(* CoDeSys 2.3.9.31 project: BA17xx.pro *)
(* Libraries: TcBaseMath.lib 27.7.04 13:07:56, TcMC2_Camming.lib 11.12.14 09:45:00, TcMath.lib 23.9.04 16:15:30, TcNC.lib 10.10.08 18:55:34, TcBase.lib 14.5.09 13:14:08, TcMC2.lib 22.12.11 16:37:48, TcSystem.lib 9.3.10 11:21:30, TcXmlDataSrv.lib 29.9.06 15:13:00, TcUtilities.lib 7.4.10 10:22:08, COMlibV2.lib 1.8.08 14:22:48, TcRFID.lib 20.9.10 12:18:58, STANDARD.LIB 5.6.98 13:03:02, TcCX1000System.lib 11.10.10 12:52:26, TcEtherCAT.lib 15.1.10 20:43:56, TcTestAndSet.lib 23.2.09 13:50:08, TcDrive.lib 17.3.10 13:50:30, TcMc2Drive.lib 19.1.10 11:34:38, TcIoFunctions.lib 21.7.11 17:19:20 *)

(* Global variable list: EPT Lib/Global_Checks *)
VAR_GLOBAL
	CheckBounds_ErrCnt 			: DINT := 0;
	CheckByteZeroDiv_ErrCnt 		: DINT := 0;
	CheckDWordZeroDiv_ErrCnt 	: DINT := 0;
	CheckRealZeroDiv_ErrCnt 		: DINT := 0;
	CheckWordZeroDiv_ErrCnt 		: DINT := 0;
	CheckRangeSigned_ErrCnt		: DINT := 0;
	CheckRangeUnsigned_ErrCnt	: DINT := 0;
END_VAR

(* Global variable list: Global_Visu *)
VAR_GLOBAL
	visu 			: 	struct_visu;
	visu_hinten	:	struct_visu_hinten;
END_VAR

(* Global variable list: Globale_Achsen *)
VAR_GLOBAL
	(* Achsen *)
	z_achse								: AXIS_REF;
	axis_z_achse							: struct_achse;

	bestueckachse						: AXIS_REF;
	axis_bestueckachse					: struct_achse;

	virtuelle_master_achse					: AXIS_REF;
	axis_virt_master						: struct_achse;

	getriebe_einstell_achse					: AXIS_REF;

	y_achse								: AXIS_REF;
	axis_y_achse							: struct_achse;

	b_achse								: AXIS_REF;
	axis_bandeinzug_achse				: struct_achse;

	transport_wt_achse					:AXIS_REF;
	axis_transport_wt_achse				: struct_achse;
END_VAR

(* Global variable list: Globale_IO *)
VAR_GLOBAL
	(* =====SMEMA -Schnittstelle===== *)
	(* Digitale IO *)
	(* SMEMA -Schnittstelle *)
	e_smema_station_vorher_in_anforderung			AT %I* : BOOL;
	e_smema_station_vorher_in_abgegeben			AT %I* : BOOL;
	a_smema_station_vorher_out_erlaubnis			AT %Q* : BOOL;
	a_smema_station_vorher_out_angekommen		AT %Q* : BOOL;

	e_smema_station_nachher_in_erlaubnis			AT %I* : BOOL;
	e_smema_station_nachher_in_angekommen		AT %I* : BOOL;
	a_smema_station_nachher_out_anforderung		AT %Q* : BOOL;
	a_smema_station_nachher_out_abgegeben		AT %Q* : BOOL;

	(* ADS-Kommunikation *)
	st_ads_smema_station_vorher					: struct_station_vorher;
	st_ads_smema_station_nachher					: struct_station_nachher;

	(* Bandwechselvorschub/Rasterfolienvorschub *)
	a_zyl_vorschub_einfahren						AT %Q* : BOOL;
	a_zyl_vorschub_ausfahren						AT %Q* : BOOL;

	(* Fänger Rasterfolie/Bandeinzug bzw. Klemmen Rasterfolie/Bandeinzug *)
	a_zyl_faenger_einfahren						AT %Q* : BOOL;
	a_zyl_klemmen_einfahren						AT %Q* : BOOL;
END_VAR

(* Global variable list: EPT Lib/Globale_Var *)
VAR_GLOBAL
	gi16_betriebsart					: enum_betriebsarten;
END_VAR

VAR_GLOBAL PERSISTENT
	gst_system_time					: TIMESTRUCT;
	gdt_system_time					: DT;
	gstr_system_time				: STRING;
	b_system_time_valid				: BOOL;
	gstr_datum						: STRING;
	gstr_uhrzeit						: STRING;
END_VAR

VAR_GLOBAL CONSTANT
	MAX_NOCKENGERUEST			: INT := 63;
END_VAR

(* Global variable list: Globale_Var_BA *)
VAR_GLOBAL
	garr_stoermeldungen				: ARRAY[0..4999] OF BOOL;
	garr_betriebsmeldungen			: ARRAY[0..4999] OF BOOL;

	gb_ba_auto_kontroller				: BOOL;
	gi16_maschinenstatusinfo			: enum_maschinenstatus;
	gb_nach_bawe_einzelfertigung		: BOOL := FALSE;
	gi16_anzahl_Teile_autostop_bandwechsel	: INT := 0;

	bbgen							: struct_objekt;
	wartung							: struct_objekt;
	bandspruehoeler					: struct_objekt;
	haspel_re						: struct_haspel_V2;
	haspel_li							: struct_haspel_V2;
	betriebsarten						: struct_betriebsarten;
	bandeinzug_kontroller				: struct_objekt;
	bandwechsel_kontroller			: struct_bandwechsler;
	haspel_kontroller					: struct_haspelkontroller;
	stoerungen_quittieren				: struct_objekt;
	betriebsfreigaben					: struct_betriebsfreigaben;
	betriebsstundenzaehler			: struct_betriebsstundenzaehler;
	wkz_absicherung					: struct_objekt;
	stueckzahlen						: struct_stueckzahl;
	balluff_tag_reader					: struct_balluff_tag_reader;
	barcode							: struct_barcode;
	hublift_links						: struct_objekt;
	hublift_rechts						: struct_objekt;
	wt_transport_kontroller				: struct_objekt;
	wt_transport_beladen				: struct_objekt;
	wt_transport_warteposition_1700		: struct_objekt;
	wt_transport_beladen_achse_1700	: struct_objekt;
	wt_transport_beladen_1720			: struct_objekt;
	wt_transport_warteposition_1720		: struct_objekt;
	wt_transport_abgabe				: struct_objekt;
	safety							: struct_objekt;
	xml_server						: struct_objekt;
	fb_edit_mfps_bestuecken_z			: struct_mf_editor;
	fb_edit_mfps_bestuecken_y			: struct_mf_editor;
	fb_edit_mfps_bestuecken_b		: struct_mf_editor;
	fb_edit_mfps_yz_tisch	 			: struct_mf_editor;
	fb_edit_mfps_bestueckachse		: struct_mf_editor;
	fb_camtable_bestueckachse		: struct_camtable_maker;
	(*rasterplattenmontage				: struct_objekt;
	rasterplattenwendestation			: struct_objekt;
	ruettler_rasterplatte				: struct_rapl_ruettler;*)
	einpresskraft_kontroller				: struct_objekt;
	kraftmessdose					: struct_analogin;
	nockenschaltwerk_bestueckachse	: struct_nockenschaltwerk_lreal;
	routing_backpanel					: struct_objekt;
	routing_nachbarpc					: struct_objekt;
	ads_kommu_pc_vorher			: struct_ads_kommunikation;
	ads_kommu_pc_nachher			: struct_ads_kommunikation;
	rasterfolienmontage				: struct_objekt;
	rasterfolieneinzug					: struct_objekt;
	edit_mfps						: struct_objekt;
	Lesen_Schreiben_Tag				: struct_objekt;
	Service							: struct_objekt;

	UPS							: struct_objekt;

	st_ctrl_in_empty					:struct_ctrl_in;
	st_ctrl_out_empty				:struct_ctrl_out;

	(* Daten welche vom Tag gelesen / zum Tag geschrieben werden *)
	gst_tag_data						: struct_tag_data;

	gi16_bbgen_auftrag				: enum_bbgen_auftrag := KEIN_BB_AUFTRAG;
	gi16_wartung_auftrag				: enum_wartung_auftrag :=  KEIN_WARTUNG_AUFTRAG;

	gst_bestueckbild					: struct_bestueckbild;
	gst_bestueckbild_halbauto			: struct_bestueckbild_halbauto;
	s_alte_artikelnummer				: STRING(50) := '';

	(* Version *)
	gs_version						: STRING := '*.zip';
	lr_debug : LREAL;

	(* Datenstruktur der Werkzeuge und STV auf der Maschine, welche per XML-File auf der Festplatte abgespeichert werden *)
	gst_datensatz						: struct_datensatz;

	(* Barcodedaten *)
	gst_barcode_daten				: struct_barcode_daten;

	gb_memEndOfBandMarkNIO		: BOOL := FALSE;	(*
	Diese Änderung wurde 1:1 aus Tschechien übernommen.
	Merker "gb_memEndOfBandMarkNIO" für Bandende während des Bestückens. Diese Variable gilt nur
	für den One27 in Tschechien. Während des Bestückens wird der Bandende Sensor abgefragt. Wenn
	noch mehr wie 80 Pins zu bestücken sind und der Bandende Sensor anschlägt, wird ein "HALT_AXIS"
	der virtuellen Masterachse ausgeführt. Die Achse bleibt zufällig irgendwo stehen. Der WT bleibt auf
	Bestückposition stehen. Eine Fehlermeldung kommt vom Bandwechselkontroller. Dann muss die 
	Anlage quittiert werden. Bestückachse fährt in Grundstellung und WT fährt auf Übergabeposition.
	Danach wird der Bandwechselvorgang gestartet. *)

	EtherCatDiag						:ARRAY[1..MaxNoOfMaster] OF FB_EtherCatDiag;
END_VAR

VAR_GLOBAL PERSISTENT
	(* manuelles Bestückbild *)
	gst_manuelles_bestueckprogramm	: struct_bestueckprogramm;
	gst_PersDaten						: struct_PD;
END_VAR
VAR_GLOBAL CONSTANT
	MaxNoOfMaster					:INT:=4;(*Maximale Anzahl Master für Ethercat Diagnose*)
	MaxNoOfSlaves					:INT:=40;(*Maximale Anzahl Slaves für Ethercat Diagnose*)
	MaxNoOfWkz						:INT:=24;(*Maximale Anzahl an Werkzeuge*)
END_VAR

(* Global variable list: Globale_XML_Server *)
VAR_GLOBAL
	(* Initialisierung der zu schreibenden Variablen in dem XML-File *)
	gs_xml_laufwerk					: STRING := 'D:\';
	gs_xml_path_root				: STRING := 'BBGen';
	gs_xml_path_md					: STRING(255) := 'MD';
	gs_xml_dateiname_md			: STRING := 'Maschinendaten';
	gs_xml_path_wkz				: STRING := 'WKZ';
	gs_xml_datei_erweiterung		: STRING := '.xml';
	gs_xml_symname_wkz			: STRING := 'gst_datensatz.st_wkz';
	gs_xml_symname_md			: STRING := 'gst_datensatz.st_md';
	s_PLC_name					: STRING(255);
	s_PLC_path						: STRING(255);
	s_Projekt_path					: STRING(255);

	(* Pfadnamen für Daten (ohne Laufwerksangabez.B."C:\_Datensatz" wird der Projektpfad angehängt)*)
	s_tools_path					: STRING(255):='Tools\';
	s_md_path 						: STRING(255):='MD\';

END_VAR

(* Global variable list: Globale_Zylinder *)
VAR_GLOBAL
	(* Gemeinsam *)
	zyl_wt_zentrierer_tisch				: struct_st_zylinder;
	zyl_wt_stopper_tisch				: struct_st_zylinder;
	zyl_wt_stopper_auslauf				: struct_st_zylinder;

	zyl_haspel_re_heben				: struct_st_zylinder;
	zyl_haspel_re_abspulen			: struct_st_zylinder;
	zyl_haspel_li_heben				: struct_st_zylinder;
	zyl_haspel_li_abspulen			: struct_st_zylinder;
	zyl_haspel_re_sperren				: struct_st_zylinder;
	zyl_haspel_li_sperren			:	 struct_st_zylinder;

	zyl_hublift_rechts_lift				: struct_st_zylinder;
	zyl_hublift_rechts_wt_einzug			: struct_st_zylinder;
	zyl_hublift_rechts_wt_klinke			: struct_st_zylinder;
	zyl_hublift_links_lift					: struct_st_zylinder;
	zyl_hublift_links_wt_einzug			: struct_st_zylinder;
	zyl_hublift_links_wt_klinke			: struct_st_zylinder;
	zyl_hublift_links_stopper			: struct_st_zylinder;
	zyl_hublift_links_eingriffschutz		: struct_st_zylinder;

	(* BSH 1700 *)
	zyl_bandfaenger					: struct_st_zylinder;
	zyl_bandklemmen					: struct_st_zylinder;
	zyl_bawe_vorschub				: struct_st_zylinder;
	zyl_bawe_querschub				: struct_st_zylinder;
	zyl_bawe_faenger_li				: struct_st_zylinder;
	zyl_bawe_faenger_re				: struct_st_zylinder;
	zyl_bawe_halter_li					: struct_st_zylinder;
	zyl_bawe_halter_re				: struct_st_zylinder;
	zyl_haspel_verschieben			: struct_st_zylinder;
	zyl_bandeinzuege_verschieben		: struct_st_zylinder;
	zyl_oelen_unten				: struct_st_zylinder;
	zyl_oelen_oben				: struct_st_zylinder;
	zyl_Indexier_Bestueckpos			: struct_st_zylinder;
	zyl_Indexier_Einlauf				: struct_st_zylinder;

	(* Rasterplatte *)
(*	zyl_rapl_aufpressen				: struct_st_zylinder;
	zyl_rapl_schacht					: struct_st_zylinder;
	zyl_rapl_kontaktfuehrung			: struct_st_zylinder;
	zyl_rap_ausschieben				: struct_st_zylinder;
	zyl_rapl_einschieben				: struct_st_zylinder;*)

	(* BSV1720 *)
	zyl_wt_stopper_einlauf				: struct_st_zylinder;
	zyl_bandfaenger_li				: struct_st_zylinder;
	zyl_bandfaenger_re				: struct_st_zylinder;
	zyl_bandklemmen_li				: struct_st_zylinder;
	zyl_bandklemmen_re				: struct_st_zylinder;

	(* Rasterfolie *)
	zyl_rafo_faenger					: struct_st_zylinder;
	zyl_rafo_klemmen					: struct_st_zylinder;
	zyl_rafo_vorschub					: struct_st_zylinder;
	zyl_rafo_kamm					: struct_st_zylinder;
	zyl_rafo_vorzentrierer				: struct_st_zylinder;
END_VAR

(* Global variable list: TwinCAT_Configuration *)
(* Generated automatically by TwinCAT - (read only) *)
VAR_CONFIG
	ST_AbfallBlasluft.a_AbfallBlasluft AT %QX5.0 : BOOL;
	ST_Bandeinzug_Kontroller_1700.e_wc_state AT %IX1272.0 : BOOL;
	ST_Bandeinzug_Kontroller_1700.e_gls_bandvorschubkontrolle AT %IX16.0 : BOOL;	(*  ~ {LinkedWith:TIID^Gerät 1 (EtherCAT)^A160 (EP2338-0001)^Channel 3^ST_Rasterfolienmontage.e_rasterfolie_aufgepresst} *)
	ST_Bandeinzug_Kontroller_1720.e_ls_bandende_re AT %IX16.1 : BOOL;
	ST_Bandeinzug_Kontroller_1720.e_ls_bandende_li AT %IX16.2 : BOOL;
	ST_Bandeinzug_Kontroller_1720.e_wc_state AT %IX1272.1 : BOOL;
	ST_Bandeinzug_Kontroller_1720.e_gls_bandvorschubkontrolle_li AT %IX820.0 : BOOL;
	ST_Bandeinzug_Kontroller_1720.e_gls_bandvorschubkontrolle_re AT %IX820.1 : BOOL;
	ST_BandoelerZylinder.a_ventil_oben AT %QX1144.0 : BOOL;	(*  ~ {LinkedWith:TIID^Gerät 1 (EtherCAT)^A170 (EP2338-0001)^Channel 15^ST_BandoelerZylinder.a_ventil_oben} *)
	ST_BandoelerZylinder.a_ventil_unten AT %QX1144.1 : BOOL;	(*  ~ {LinkedWith:TIID^Gerät 1 (EtherCAT)^A170 (EP2338-0001)^Channel 16^ST_BandoelerZylinder.a_ventil_unten} *)
	ST_BandoelerZylinder.e_fuellstand AT %IX1280.0 : BOOL;	(*  ~ {LinkedWith:TIID^Gerät 1 (EtherCAT)^A38 Transportsystem (EP2338-0001)^Channel 8^ST_Menzel_Spruehoeler.e_fuellstand} *)
	ST_BandoelerZylinder.e_druck_oelbehaelter AT %IX1280.1 : BOOL;	(*  ~ {LinkedWith:TIID^Gerät 1 (EtherCAT)^A38 Transportsystem (EP2338-0001)^Channel 7^ST_Menzel_Spruehoeler.e_druck_oelbehaelter} *)
	ST_Bandwechsel_Kontroller.e_ls_bandende_li AT %IX16.4 : BOOL;	(*  ~ {LinkedWith:TIID^Gerät 1 (EtherCAT)^A150 (EP2338-0001)^Channel 3^ST_Bandwechsel_Kontroller.e_ls_bandende_li} *)
	ST_Bandwechsel_Kontroller.e_ls_bandende_re AT %IX16.5 : BOOL;	(*  ~ {LinkedWith:TIID^Gerät 1 (EtherCAT)^A150 (EP2338-0001)^Channel 4^ST_Bandwechsel_Kontroller.e_ls_bandende_re} *)
	ST_Bestueckachse.fb_axis.e_limit_sensor_positive AT %IX30.5 : BOOL;
	ST_Bestueckachse.fb_axis.e_limit_sensor_negative AT %IX30.6 : BOOL;
	ST_Bestueckachse.fb_axis.e_referenz_sensor AT %IX30.7 : BOOL;
	ST_Bestueckachse.e_referenz_sensor AT %IX16.6 : BOOL;	(*  ~ {LinkedWith:TIID^Gerät 1 (EtherCAT)^Schaltschrank (EK1100)^A32 (EL1819)^Channel 8^ST_Bestueckachse.e_referenz_sensor} *)
	ST_Bestueckachse.i16_torque AT %IB0 : INT;
	ST_Betriebsarten.e_ba_automatik AT %IX16.7 : BOOL;	(*  ~ {LinkedWith:TIID^Gerät 1 (EtherCAT)^Schaltschrank (EK1100)^A17 (EL6900)^Module 2 (FSOE)^Standard Out Vars TxPDO 1^Standard Out Var 4} *)
	ST_Betriebsarten.e_ba_tippen AT %IX17.0 : BOOL;	(*  ~ {LinkedWith:TIID^Gerät 1 (EtherCAT)^Schaltschrank (EK1100)^A17 (EL6900)^Module 2 (FSOE)^Standard Out Vars TxPDO 1^Standard Out Var 5} *)
	ST_Betriebsarten.e_ba_hand AT %IX17.1 : BOOL;	(*  ~ {LinkedWith:TIID^Gerät 1 (EtherCAT)^Schaltschrank (EK1100)^A17 (EL6900)^Module 2 (FSOE)^Standard Out Vars TxPDO 1^Standard Out Var 6} *)
	ST_Betriebsarten.e_ba_dummy AT %IX17.2 : BOOL;
	ST_Betriebsarten.e_ba_pseudo AT %IX17.3 : BOOL;
	ST_Betriebsarten.a_lampe_ba_automatik AT %QX5.1 : BOOL;
	ST_Betriebsarten.a_lampe_ba_tippen AT %QX5.2 : BOOL;
	ST_Betriebsarten.a_lampe_ba_hand AT %QX5.3 : BOOL;
	ST_Betriebsarten.a_lampe_ba_dummy AT %QX5.4 : BOOL;
	ST_Betriebsarten.a_lampe_ba_pseudo AT %QX5.5 : BOOL;
	ST_Betriebsfreigaben.e_temperatur_schaltschrank AT %IX17.4 : BOOL;	(*  ~ {LinkedWith:TIID^Gerät 1 (EtherCAT)^Schaltschrank (EK1100)^A31 (EL1819)^Channel 2^ST_Betriebsfreigaben.e_temperatur_schaltschrank} *)
	ST_Betriebsfreigaben.e_ls_schalter_ausgeloest AT %IX17.5 : BOOL;	(*  ~ {LinkedWith:TIID^Gerät 1 (EtherCAT)^Schaltschrank (EK1100)^A31 (EL1819)^Channel 1^ST_Betriebsfreigaben.e_ls_schalter_ausgeloest} *)
	ST_Betriebsfreigaben.e_ueberstrom_haspel AT %IX18.0 : BOOL;	(*  ~ {LinkedWith:TIID^Gerät 1 (EtherCAT)^Schaltschrank (EK1100)^A31 (EL1819)^Channel 4^ST_Betriebsfreigaben.e_ueberstrom_haspel} *)
	ST_Betriebsfreigaben.a_lampe_steuerung AT %QX5.6 : BOOL;	(*  ~ {LinkedWith:TIID^Gerät 1 (EtherCAT)^Schaltschrank (EK1100)^A46 (EL2809)^Channel 1^ST_Betriebsfreigaben.a_lampe_steuerung} *)
	ST_Betriebsfreigaben.e_druckwaechter AT %IX18.1 : BOOL;	(*  ~ {LinkedWith:TIID^Gerät 1 (EtherCAT)^Schaltschrank (EK1100)^A31 (EL1819)^Channel 3^ST_Betriebsfreigaben.e_druckwaechter} *)
	ST_Betriebsfreigaben.e_druckwaechter_hublift_links AT %IX1280.2 : BOOL;	(*  ~ {LinkedWith:TIID^Gerät 1 (EtherCAT)^A200 Hublift Links (EK1101)^A201 (EL1819)^Channel 14^ST_Betriebsfreigaben.e_druckwaechter_hublift_links} *)
	ST_Betriebsfreigaben.a_lampe_stoerung AT %QX5.7 : BOOL;	(*  ~ {LinkedWith:TIID^Gerät 1 (EtherCAT)^Schaltschrank (EK1100)^A46 (EL2809)^Channel 3^ST_Betriebsfreigaben.a_lampe_stoerung} *)
	ST_Betriebsfreigaben.a_lampe_produktion AT %QX6.0 : BOOL;	(*  ~ {LinkedWith:TIID^Gerät 1 (EtherCAT)^Schaltschrank (EK1100)^A46 (EL2809)^Channel 5^ST_Betriebsfreigaben.a_lampe_produktion} *)
	ST_Einpress_Kontroller.a_start_messung AT %QX6.1 : BOOL;	(*  ~ {LinkedWith:TIID^Gerät 1 (EtherCAT)^Schaltschrank (EK1100)^A47 (EL2809)^Channel 3^ST_Einpress_Kontroller.a_start_messung} *)
	ST_Einpress_Kontroller.a_messbereich_1_oder_2 AT %QX6.2 : BOOL;	(*  ~ {LinkedWith:TIID^Gerät 1 (EtherCAT)^Schaltschrank (EK1100)^A47 (EL2809)^Channel 4^ST_Einpress_Kontroller.a_messbereich_1_oder_2} *)
	ST_EthercatDiag.arr_ec_slave_net_id AT %IB824 : ARRAY [0..8] OF T_AmsNetIdArr;
	ST_Euchner_Handbedienpult.e_Taste_Zustimm AT %IX18.2 : BOOL;
	ST_Euchner_Handbedienpult.e_Taste_Plus AT %IX18.3 : BOOL;	(*  ~ {LinkedWith:TIID^Gerät 1 (EtherCAT)^Schaltschrank (EK1100)^A31 (EL1819)^Channel 16^ST_Euchner_Handbedienpult.e_Taste_Plus} *)
	ST_Euchner_Handbedienpult.e_Taste_Power AT %IX18.4 : BOOL;	(*  ~ {LinkedWith:TIID^Gerät 1 (EtherCAT)^Schaltschrank (EK1100)^A31 (EL1819)^Channel 15^ST_Euchner_Handbedienpult.e_Taste_Power} *)
	ST_Euchner_Handbedienpult.e_Taste_Minus AT %IX18.5 : BOOL;	(*  ~ {LinkedWith:TIID^Gerät 1 (EtherCAT)^Schaltschrank (EK1100)^A31 (EL1819)^Channel 14^ST_Euchner_Handbedienpult.e_Taste_Minus} *)
	ST_Euchner_Handbedienpult.e_i16_Zaehler AT %IB2 : INT;	(*  ~ {LinkedWith:TIID^Gerät 1 (EtherCAT)^Schaltschrank (EK1100)^A41 (EL5101)^ENC Status compact^Counter value} *)
	ST_Gesamthubzaehler.a_Gesamthubzaehler AT %QX6.3 : BOOL;	(*  ~ {LinkedWith:TIID^Gerät 1 (EtherCAT)^Schaltschrank (EK1100)^A46 (EL2809)^Channel 16^ST_Gesamthubzaehler.a_Gesamthubzaehler} *)
	ST_Haspel_Kontroller_2H.e_haspelmotor_bb AT %IX18.6 : BOOL;
	ST_Haspel_Kontroller_2H.a_motor_drehrichtung_rechts AT %QX6.4 : BOOL;	(*  ~ {LinkedWith:TIID^Gerät 1 (EtherCAT)^Schaltschrank (EK1100)^A46 (EL2809)^Channel 7^ST_Haspel_Kontroller_2H.a_motor_drehrichtung_rechts} *)
	ST_Haspel_Kontroller_2H.a_motor_drehrichtung_links AT %QX6.5 : BOOL;	(*  ~ {LinkedWith:TIID^Gerät 1 (EtherCAT)^Schaltschrank (EK1100)^A46 (EL2809)^Channel 6^ST_Haspel_Kontroller_2H.a_motor_drehrichtung_links} *)
	ST_Hublift_links.e_sensor_wt_anwesend AT %IX18.7 : BOOL;	(*  ~ {LinkedWith:TIID^Gerät 1 (EtherCAT)^A200 Hublift Links (EK1101)^A201 (EL1819)^Channel 9^ST_Hublift_links.e_sensor_wt_anwesend} *)
	ST_Hublift_links.e_sensor_wt_von_fb_eingezogen AT %IX19.0 : BOOL;	(*  ~ {LinkedWith:TIID^Gerät 1 (EtherCAT)^A200 Hublift Links (EK1101)^A201 (EL1819)^Channel 10^ST_Hublift_links.e_sensor_wt_von_fb_eingezogen} *)
	ST_Hublift_links.e_wc_state AT %IX1272.2 : BOOL;	(*  ~ {LinkedWith:TIID^Gerät 1 (EtherCAT)^A200 Hublift Links (EK1101)^WcState^WcState} *)
	ST_Hublift_links.e_schiebetuere_geschlossen AT %IX1280.3 : BOOL;	(*  ~ {LinkedWith:TIID^Gerät 1 (EtherCAT)^A200 Hublift Links (EK1101)^A201 (EL1819)^Channel 16^ST_Hublift_links.e_schiebetuere_geschlossen} *)
	ST_Hublift_links.a_lampe_erlaubnis_schiebetuere_oeffnen AT %QX1144.2 : BOOL;	(*  ~ {LinkedWith:TIID^Gerät 1 (EtherCAT)^A200 Hublift Links (EK1101)^A203 (EL2809)^Channel 13^ST_Hublift_links.a_lampe_erlaubnis_schiebetuere_oeffnen} *)
	ST_Hublift_rechts.e_sensor_wt_anwesend AT %IX19.1 : BOOL;	(*  ~ {LinkedWith:TIID^Gerät 1 (EtherCAT)^A250 Hublift Rechts (EK1101)^A251 (EL1819)^Channel 9^ST_Hublift_rechts.e_sensor_wt_anwesend} *)
	ST_Hublift_rechts.e_wc_state AT %IX1272.3 : BOOL;
	ST_LampeMaterialMangel.a_Lampe AT %QX6.6 : BOOL;	(*  ~ {LinkedWith:TIID^Gerät 1 (EtherCAT)^Schaltschrank (EK1100)^A46 (EL2809)^Channel 4^ST_LampeMaterialMangel.a_Lampe} *)
	ST_Menzel_Spruehoeler.a_ventil AT %QX6.7 : BOOL;	(*  ~ {LinkedWith:TIID^Gerät 1 (EtherCAT)^Schaltschrank (EK1100)^A46 (EL2809)^Channel 9^ST_Menzel_Spruehoeler.a_ventil} *)
	ST_Menzel_Spruehoeler.e_fuellstand AT %IX19.2 : BOOL;	(*  ~ {LinkedWith:TIID^Gerät 1 (EtherCAT)^A38 Transportsystem (EP2338-0001)^Channel 8^ST_Menzel_Spruehoeler.e_fuellstand} *)
	ST_Menzel_Spruehoeler.e_druck_oelbehaelter AT %IX19.3 : BOOL;	(*  ~ {LinkedWith:TIID^Gerät 1 (EtherCAT)^A38 Transportsystem (EP2338-0001)^Channel 7^ST_Menzel_Spruehoeler.e_druck_oelbehaelter} *)
	ST_Rasterfolieneinzug.e_rasfo_ende AT %IX19.5 : BOOL;	(*  ~ {LinkedWith:TIID^Gerät 1 (EtherCAT)^A150 (EP2338-0001)^Channel 3^ST_Bandwechsel_Kontroller.e_ls_bandende_li} *)
	ST_Rasterfolieneinzug.e_rasfo_vorschubkontrolle AT %IX19.6 : BOOL;	(*  ~ {LinkedWith:TIID^Gerät 1 (EtherCAT)^A150 (EP2338-0001)^Channel 4^ST_Bandwechsel_Kontroller.e_ls_bandende_re} *)
	ST_Rasterfolieneinzug.e_rasfo_rueckzugueberwachung AT %IX19.7 : BOOL;	(*  ~ {LinkedWith:TIID^Gerät 1 (EtherCAT)^A160 (EP2338-0001)^Channel 3^ST_Rasterfolienmontage.e_rasterfolie_aufgepresst} *)
	ST_Rasterfolieneinzug.aIonisierungEin AT %QX1308.0 : BOOL;
	ST_Rasterfolienmontage.e_rasterfolie_aufgepresst AT %IX20.0 : BOOL;	(*  ~ {LinkedWith:TIID^Gerät 1 (EtherCAT)^A160 (EP2338-0001)^Channel 3^ST_Rasterfolienmontage.e_rasterfolie_aufgepresst} *)
	ST_Safetyprogramm.a_quitt_pilz_hublift_links AT %QX1144.4 : BOOL;	(*  ~ {LinkedWith:TIID^Gerät 1 (EtherCAT)^A200 Hublift Links (EK1101)^A205 (EL2809)^Channel 1^ST_Safetyprogramm.a_quitt_pilz_hublift_links} *)
	ST_Safetyprogramm.a_lampe_quitt_schutztuere_vorne AT %QX7.1 : BOOL;	(*  ~ {LinkedWith:TIID^Gerät 1 (EtherCAT)^Schaltschrank (EK1100)^A46 (EL2809)^Channel 2^ST_Safetyprogramm.a_lampe_quitt_schutztuere_vorne} *)
	ST_Safetyprogramm.a_lampe_quitt_schutztuere_hinten AT %QX7.2 : BOOL;	(*  ~ {LinkedWith:TIID^Gerät 1 (EtherCAT)^Schaltschrank (EK1100)^A47 (EL2809)^Channel 7^ST_Safetyprogramm.a_lampe_quitt_schutztuere_hinten} *)
	ST_Safetyprogramm.se_quittiertaste AT %IX20.5 : BOOL;	(*  ~ {LinkedWith:TIID^Gerät 1 (EtherCAT)^Schaltschrank (EK1100)^A17 (EL6900)^Module 2 (FSOE)^Standard Out Vars TxPDO 1^Standard Out Var 7} *)
	ST_Safetyprogramm.se_taste_steuerung_ein AT %IX1268.0 : BOOL;	(*  ~ {LinkedWith:TIID^Gerät 1 (EtherCAT)^Schaltschrank (EK1100)^A17 (EL6900)^Module 2 (FSOE)^Standard Out Vars TxPDO 1^ST_Safetyprogramm.se_taste_steuerung_ein} *)
	ST_Safetyprogramm.se_taste_steuerung_aus AT %IX1268.1 : BOOL;	(*  ~ {LinkedWith:TIID^Gerät 1 (EtherCAT)^Schaltschrank (EK1100)^A17 (EL6900)^Module 2 (FSOE)^Standard Out Vars TxPDO 1^ST_Safetyprogramm.se_taste_steuerung_aus} *)
	ST_Safetyprogramm.se_steuerung_ein AT %IX20.6 : BOOL;	(*  ~ {LinkedWith:TIID^Gerät 1 (EtherCAT)^Schaltschrank (EK1100)^A17 (EL6900)^Module 2 (FSOE)^Standard Out Vars TxPDO 1^Standard Out Var 12} *)
	ST_Safetyprogramm.se_ba_mit_bedingungen AT %IX20.7 : BOOL;	(*  ~ {LinkedWith:TIID^Gerät 1 (EtherCAT)^Schaltschrank (EK1100)^A17 (EL6900)^Module 2 (FSOE)^Standard Out Vars TxPDO 1^Standard Out Var 13} *)
	ST_Safetyprogramm.se_nothalt_gesamt_ok AT %IX21.0 : BOOL;	(*  ~ {LinkedWith:TIID^Gerät 1 (EtherCAT)^Schaltschrank (EK1100)^A17 (EL6900)^Module 2 (FSOE)^Standard Out Vars TxPDO 1^Standard Out Var 11} *)
	ST_Safetyprogramm.se_tuere_vorne_diskrepanz AT %IX21.1 : BOOL;	(*  ~ {LinkedWith:TIID^Gerät 1 (EtherCAT)^Schaltschrank (EK1100)^A17 (EL6900)^Module 2 (FSOE)^Standard Out Vars TxPDO 1^Standard Out Var 15} *)
	ST_Safetyprogramm.se_tuere_hinten_diskrepanz AT %IX21.2 : BOOL;	(*  ~ {LinkedWith:TIID^Gerät 1 (EtherCAT)^Schaltschrank (EK1100)^A17 (EL6900)^Module 2 (FSOE)^Standard Out Vars TxPDO 1^Standard Out Var 16} *)
	ST_Safetyprogramm.se_not_halt_intern AT %IX21.3 : BOOL;	(*  ~ {LinkedWith:TIID^Gerät 1 (EtherCAT)^Schaltschrank (EK1100)^A17 (EL6900)^Module 2 (FSOE)^Standard Out Vars TxPDO 1^Standard Out Var 14} *)
	ST_Safetyprogramm.se_not_halt_frontseite AT %IX21.4 : BOOL;	(*  ~ {LinkedWith:TIID^Gerät 1 (EtherCAT)^Schaltschrank (EK1100)^A17 (EL6900)^Module 2 (FSOE)^Standard Out Vars TxPDO 1^Standard Out Var 24} *)
	ST_Safetyprogramm.se_not_halt_rueckseite AT %IX21.5 : BOOL;	(*  ~ {LinkedWith:TIID^Gerät 1 (EtherCAT)^Schaltschrank (EK1100)^A17 (EL6900)^Module 2 (FSOE)^Standard Out Vars TxPDO 1^Standard Out Var 25} *)
	ST_Safetyprogramm.se_not_halt_bediengeraet AT %IX21.6 : BOOL;	(*  ~ {LinkedWith:TIID^Gerät 1 (EtherCAT)^Schaltschrank (EK1100)^A17 (EL6900)^Module 2 (FSOE)^Standard Out Vars TxPDO 1^Standard Out Var 26} *)
	ST_Safetyprogramm.se_not_halt_extern AT %IX21.7 : BOOL;	(*  ~ {LinkedWith:TIID^Gerät 1 (EtherCAT)^Schaltschrank (EK1100)^A17 (EL6900)^Module 2 (FSOE)^Standard Out Vars TxPDO 1^Standard Out Var 23} *)
	ST_Safetyprogramm.se_tuere_vorne_offen AT %IX22.0 : BOOL;	(*  ~ {LinkedWith:TIID^Gerät 1 (EtherCAT)^Schaltschrank (EK1100)^A17 (EL6900)^Module 2 (FSOE)^Standard Out Vars TxPDO 1^Standard Out Var 17} *)
	ST_Safetyprogramm.se_tuere_hinten_offen AT %IX22.1 : BOOL;	(*  ~ {LinkedWith:TIID^Gerät 1 (EtherCAT)^Schaltschrank (EK1100)^A17 (EL6900)^Module 2 (FSOE)^Standard Out Vars TxPDO 1^Standard Out Var 18} *)
	ST_Safetyprogramm.se_tuere_zustimm_vorne_offen AT %IX22.2 : BOOL;	(*  ~ {LinkedWith:TIID^Gerät 1 (EtherCAT)^Schaltschrank (EK1100)^A17 (EL6900)^Module 2 (FSOE)^Standard Out Vars TxPDO 1^Standard Out Var 27} *)
	ST_Safetyprogramm.se_tuere_zustimm_hinten_offen AT %IX22.3 : BOOL;	(*  ~ {LinkedWith:TIID^Gerät 1 (EtherCAT)^Schaltschrank (EK1100)^A17 (EL6900)^Module 2 (FSOE)^Standard Out Vars TxPDO 1^Standard Out Var 28} *)
	ST_Safetyprogramm.se_bestueckachse_sto AT %IX22.4 : BOOL;
	ST_Safetyprogramm.se_bestueckachse_sls AT %IX22.5 : BOOL;
	ST_Safetyprogramm.se_z_achse_sto AT %IX22.6 : BOOL;
	ST_Safetyprogramm.se_z_achse_sls AT %IX22.7 : BOOL;
	ST_Safetyprogramm.se_y_achse_sto AT %IX23.0 : BOOL;
	ST_Safetyprogramm.se_y_achse_sls AT %IX23.1 : BOOL;
	ST_Safetyprogramm.se_b_achse_sto AT %IX880.0 : BOOL;
	ST_Safetyprogramm.se_b_achse_sls AT %IX880.1 : BOOL;
	ST_Safetyprogramm.se_transport_achse_sto AT %IX1446.0 : BOOL;
	ST_Safetyprogramm.se_transport_achse_sls AT %IX1446.1 : BOOL;
	ST_Safetyprogramm.e_not_halt_hublift_links_ok AT %IX1280.6 : BOOL;	(*  ~ {LinkedWith:TIID^Gerät 1 (EtherCAT)^A200 Hublift Links (EK1101)^A201 (EL1819)^Channel 15^ST_Safetyprogramm.e_not_halt_hublift_links_ok} *)
	ST_Safetyprogramm.se_fehler_fb1_opmode AT %IX23.4 : BOOL;	(*  ~ {LinkedWith:TIID^Gerät 1 (EtherCAT)^Schaltschrank (EK1100)^A17 (EL6900)^Module 2 (FSOE)^Standard Out Vars TxPDO 1^Standard Out Var 22} *)
	ST_Safetyprogramm.se_fehler_fb9_estop_nothalt_front AT %IX23.5 : BOOL;	(*  ~ {LinkedWith:TIID^Gerät 1 (EtherCAT)^Schaltschrank (EK1100)^A17 (EL6900)^Module 2 (FSOE)^Standard Out Vars TxPDO 1^Standard Out Var 29} *)
	ST_Safetyprogramm.se_fehler_fb10_estop_nothalt_ext AT %IX23.6 : BOOL;	(*  ~ {LinkedWith:TIID^Gerät 1 (EtherCAT)^Schaltschrank (EK1100)^A17 (EL6900)^Module 2 (FSOE)^Standard Out Vars TxPDO 1^Standard Out Var 30} *)
	ST_Safetyprogramm.se_fehler_fb15_edm_nothalt_ext AT %IX23.7 : BOOL;	(*  ~ {LinkedWith:TIID^Gerät 1 (EtherCAT)^Schaltschrank (EK1100)^A17 (EL6900)^Module 2 (FSOE)^Standard Out Vars TxPDO 1^Standard Out Var 31} *)
	ST_Safetyprogramm.se_fehler_fb16_edm_nothalt_schuetz AT %IX24.0 : BOOL;	(*  ~ {LinkedWith:TIID^Gerät 1 (EtherCAT)^Schaltschrank (EK1100)^A17 (EL6900)^Module 2 (FSOE)^Standard Out Vars TxPDO 1^Standard Out Var 32} *)
	ST_Safetyprogramm.se_fehler_fb17_edm_ventilinsel AT %IX24.1 : BOOL;	(*  ~ {LinkedWith:TIID^Gerät 1 (EtherCAT)^Schaltschrank (EK1100)^A17 (EL6900)^Module 2 (FSOE)^Standard Out Vars TxPDO 1^Standard Out Var 33} *)
	ST_Safetyprogramm.se_fehler_fb28_edm_foerderband AT %IX24.2 : BOOL;
	ST_Safetyprogramm.se_fehler_fb30_estop_rueck AT %IX24.3 : BOOL;	(*  ~ {LinkedWith:TIID^Gerät 1 (EtherCAT)^Schaltschrank (EK1100)^A17 (EL6900)^Module 2 (FSOE)^Standard Out Vars TxPDO 1^Standard Out Var 34} *)
	ST_Safetyprogramm.se_fehler_fb31_estop_bedien AT %IX24.4 : BOOL;	(*  ~ {LinkedWith:TIID^Gerät 1 (EtherCAT)^Schaltschrank (EK1100)^A17 (EL6900)^Module 2 (FSOE)^Standard Out Vars TxPDO 1^Standard Out Var 35} *)
	ST_Safetyprogramm.se_fehler_fb35_mon_tuere_vo AT %IX24.5 : BOOL;	(*  ~ {LinkedWith:TIID^Gerät 1 (EtherCAT)^Schaltschrank (EK1100)^A17 (EL6900)^Module 2 (FSOE)^Standard Out Vars TxPDO 1^Standard Out Var 36} *)
	ST_Safetyprogramm.se_fehler_fb36_mon_tuere_hi AT %IX24.6 : BOOL;	(*  ~ {LinkedWith:TIID^Gerät 1 (EtherCAT)^Schaltschrank (EK1100)^A17 (EL6900)^Module 2 (FSOE)^Standard Out Vars TxPDO 1^Standard Out Var 37} *)
	ST_Safetyprogramm.se_fehler_fb37_mon_tuere_disk_vo AT %IX24.7 : BOOL;	(*  ~ {LinkedWith:TIID^Gerät 1 (EtherCAT)^Schaltschrank (EK1100)^A17 (EL6900)^Module 2 (FSOE)^Standard Out Vars TxPDO 1^Standard Out Var 38} *)
	ST_Safetyprogramm.se_fehler_fb38_mon_tuere_disk_hi AT %IX25.0 : BOOL;	(*  ~ {LinkedWith:TIID^Gerät 1 (EtherCAT)^Schaltschrank (EK1100)^A17 (EL6900)^Module 2 (FSOE)^Standard Out Vars TxPDO 1^Standard Out Var 39} *)
	ST_Safetyprogramm.se_fehler_fb39_mon_tuere_meld_vo AT %IX25.1 : BOOL;	(*  ~ {LinkedWith:TIID^Gerät 1 (EtherCAT)^Schaltschrank (EK1100)^A17 (EL6900)^Module 2 (FSOE)^Standard Out Vars TxPDO 1^Standard Out Var 40} *)
	ST_Safetyprogramm.se_fehler_fb40_mon_tuere_meld_hi AT %IX25.2 : BOOL;	(*  ~ {LinkedWith:TIID^Gerät 1 (EtherCAT)^Schaltschrank (EK1100)^A17 (EL6900)^Module 2 (FSOE)^Standard Out Vars TxPDO 1^Standard Out Var 41} *)
	ST_Safetyprogramm.sa_run_stop_gruppe1 AT %QX7.3 : BOOL;	(*  ~ {LinkedWith:TIID^Gerät 1 (EtherCAT)^Schaltschrank (EK1100)^A17 (EL6900)^Module 1 (FSOE)^Standard In Vars RxPDO 1^Standard In Var 1} *)
	ST_Safetyprogramm.sa_err_ack_gruppe1 AT %QX7.4 : BOOL;	(*  ~ {LinkedWith:TIID^Gerät 1 (EtherCAT)^Schaltschrank (EK1100)^A17 (EL6900)^Module 1 (FSOE)^Standard In Vars RxPDO 1^Standard In Var 2} *)
	ST_Safetyprogramm.se_fb_error_gruppe1 AT %IX25.3 : BOOL;	(*  ~ {LinkedWith:TIID^Gerät 1 (EtherCAT)^Schaltschrank (EK1100)^A17 (EL6900)^Module 2 (FSOE)^Standard Out Vars TxPDO 1^Standard Out Var 1} *)
	ST_Safetyprogramm.se_com_error_gruppe1 AT %IX25.4 : BOOL;	(*  ~ {LinkedWith:TIID^Gerät 1 (EtherCAT)^Schaltschrank (EK1100)^A17 (EL6900)^Module 2 (FSOE)^Standard Out Vars TxPDO 1^Standard Out Var 2} *)
	ST_Safetyprogramm.se_out_error_gruppe1 AT %IX25.5 : BOOL;	(*  ~ {LinkedWith:TIID^Gerät 1 (EtherCAT)^Schaltschrank (EK1100)^A17 (EL6900)^Module 2 (FSOE)^Standard Out Vars TxPDO 1^Standard Out Var 3} *)
	ST_Safetyprogramm.sa_run_stop_gruppe2 AT %QX7.5 : BOOL;	(*  ~ {LinkedWith:TIID^Gerät 1 (EtherCAT)^Schaltschrank (EK1100)^A17 (EL6900)^Module 1 (FSOE)^Standard In Vars RxPDO 1^Standard In Var 3} *)
	ST_Safetyprogramm.sa_err_ack_gruppe2 AT %QX7.6 : BOOL;	(*  ~ {LinkedWith:TIID^Gerät 1 (EtherCAT)^Schaltschrank (EK1100)^A17 (EL6900)^Module 1 (FSOE)^Standard In Vars RxPDO 1^Standard In Var 4} *)
	ST_Safetyprogramm.se_fb_error_gruppe2 AT %IX25.6 : BOOL;	(*  ~ {LinkedWith:TIID^Gerät 1 (EtherCAT)^Schaltschrank (EK1100)^A17 (EL6900)^Module 2 (FSOE)^Standard Out Vars TxPDO 1^Standard Out Var 8} *)
	ST_Safetyprogramm.se_com_error_gruppe2 AT %IX25.7 : BOOL;	(*  ~ {LinkedWith:TIID^Gerät 1 (EtherCAT)^Schaltschrank (EK1100)^A17 (EL6900)^Module 2 (FSOE)^Standard Out Vars TxPDO 1^Standard Out Var 9} *)
	ST_Safetyprogramm.se_out_error_gruppe2 AT %IX26.0 : BOOL;	(*  ~ {LinkedWith:TIID^Gerät 1 (EtherCAT)^Schaltschrank (EK1100)^A17 (EL6900)^Module 2 (FSOE)^Standard Out Vars TxPDO 1^Standard Out Var 10} *)
	ST_Safetyprogramm.sa_run_stop_gruppe3 AT %QX7.7 : BOOL;	(*  ~ {LinkedWith:TIID^Gerät 1 (EtherCAT)^Schaltschrank (EK1100)^A17 (EL6900)^Module 1 (FSOE)^Standard In Vars RxPDO 1^Standard In Var 5} *)
	ST_Safetyprogramm.sa_err_ack_gruppe3 AT %QX8.0 : BOOL;	(*  ~ {LinkedWith:TIID^Gerät 1 (EtherCAT)^Schaltschrank (EK1100)^A17 (EL6900)^Module 1 (FSOE)^Standard In Vars RxPDO 1^Standard In Var 6} *)
	ST_Safetyprogramm.se_fb_error_gruppe3 AT %IX26.1 : BOOL;	(*  ~ {LinkedWith:TIID^Gerät 1 (EtherCAT)^Schaltschrank (EK1100)^A17 (EL6900)^Module 2 (FSOE)^Standard Out Vars TxPDO 1^Standard Out Var 19} *)
	ST_Safetyprogramm.se_com_error_gruppe3 AT %IX26.2 : BOOL;	(*  ~ {LinkedWith:TIID^Gerät 1 (EtherCAT)^Schaltschrank (EK1100)^A17 (EL6900)^Module 2 (FSOE)^Standard Out Vars TxPDO 1^Standard Out Var 20} *)
	ST_Safetyprogramm.se_out_error_gruppe3 AT %IX26.3 : BOOL;	(*  ~ {LinkedWith:TIID^Gerät 1 (EtherCAT)^Schaltschrank (EK1100)^A17 (EL6900)^Module 2 (FSOE)^Standard Out Vars TxPDO 1^Standard Out Var 21} *)
	ST_Safetyprogramm.sa_run_stop_gruppe4 AT %QX8.1 : BOOL;
	ST_Safetyprogramm.sa_err_ack_gruppe4 AT %QX8.2 : BOOL;
	ST_Safetyprogramm.se_fb_error_gruppe4 AT %IX26.4 : BOOL;
	ST_Safetyprogramm.se_com_error_gruppe4 AT %IX26.5 : BOOL;
	ST_Safetyprogramm.se_out_error_gruppe4 AT %IX26.6 : BOOL;
	ST_Servobandeinzug.fb_axis.e_limit_sensor_positive AT %IX880.6 : BOOL;
	ST_Servobandeinzug.fb_axis.e_limit_sensor_negative AT %IX880.7 : BOOL;
	ST_Servobandeinzug.fb_axis.e_referenz_sensor AT %IX881.0 : BOOL;
	ST_Servobandeinzug.e_limit_sensor_positive AT %IX880.2 : BOOL;
	ST_Servobandeinzug.e_limit_sensor_negative AT %IX880.3 : BOOL;
	ST_Servobandeinzug.e_gls_bandreferenzieren AT %IX880.4 : BOOL;
	ST_Servobandeinzug.i16_torque AT %IB878 : INT;
	ST_Servobandeinzug.i16_vorgabe_stromlimit AT %QB752 : INT;
	ST_Tuerverriegelung.a_tuerverriegelung_vorne AT %QX8.3 : BOOL;	(*  ~ {LinkedWith:TIID^Gerät 1 (EtherCAT)^Schaltschrank (EK1100)^A47 (EL2809)^Channel 1^ST_Tuerverriegelung.a_tuerverriegelung_vorne} *)
	ST_Tuerverriegelung.a_tuerverriegelung_hinten AT %QX8.4 : BOOL;	(*  ~ {LinkedWith:TIID^Gerät 1 (EtherCAT)^Schaltschrank (EK1100)^A47 (EL2809)^Channel 2^ST_Tuerverriegelung.a_tuerverriegelung_hinten} *)
	ST_Tuerverriegelung.e_kontakt_tuerverriegelung_vorne AT %IX26.7 : BOOL;	(*  ~ {LinkedWith:TIID^Gerät 1 (EtherCAT)^Schaltschrank (EK1100)^A31 (EL1819)^Channel 9^ST_Tuerverriegelung.e_kontakt_tuerverriegelung_vorne} *)
	ST_Tuerverriegelung.e_kontakt_tuerverriegelung_hinten AT %IX27.0 : BOOL;	(*  ~ {LinkedWith:TIID^Gerät 1 (EtherCAT)^Schaltschrank (EK1100)^A31 (EL1819)^Channel 10^ST_Tuerverriegelung.e_kontakt_tuerverriegelung_hinten} *)
	ST_Virtuelle_Masterachse.fb_virt_master_axis.e_limit_sensor_positive AT %IX881.1 : BOOL;
	ST_Virtuelle_Masterachse.fb_virt_master_axis.e_limit_sensor_negative AT %IX881.2 : BOOL;
	ST_Virtuelle_Masterachse.fb_virt_master_axis.e_referenz_sensor AT %IX881.3 : BOOL;
	ST_WkzAbsicherung.e_wkz_sicherung_niederhalter_li AT %IX27.1 : BOOL;
	ST_WkzAbsicherung.e_wkz_sicherung_faenger_li AT %IX27.2 : BOOL;
	ST_WkzAbsicherung.e_wkz_sicherung_abfallpodest_li AT %IX27.3 : BOOL;
	ST_WkzAbsicherung.e_wkz_sicherung_niederhalter_re AT %IX27.4 : BOOL;
	ST_WkzAbsicherung.e_wkz_sicherung_faenger_re AT %IX27.5 : BOOL;
	ST_WkzAbsicherung.e_wkz_sicherung_abfallpodest_re AT %IX27.6 : BOOL;
	ST_WkzAbsicherung.e_kodierung_alt_wkz AT %IX27.7 : BOOL;
	ST_WkzAbsicherung.e_wkz_sicherung_faenger AT %IX28.0 : BOOL;	(*  ~ {LinkedWith:TIID^Gerät 1 (EtherCAT)^Schaltschrank (EK1100)^A32 (EL1819)^Channel 1^ST_WkzAbsicherung.e_wkz_sicherung_faenger} *)
	ST_WkzAbsicherung.e_bestueckschieber_ueberwachung AT %IX28.1 : BOOL;	(*  ~ {LinkedWith:TIID^Gerät 1 (EtherCAT)^Schaltschrank (EK1100)^A32 (EL1819)^Channel 6^ST_WkzAbsicherung.e_bestueckschieber_ueberwachung} *)
	ST_WT_Transport_Abgabe.e_wt_auf_abgabepos AT %IX28.2 : BOOL;	(*  ~ {LinkedWith:TIID^Gerät 1 (EtherCAT)^Schaltschrank (EK1100)^A32 (EL1819)^Channel 11^ST_WT_Transport_Abgabe.e_wt_auf_abgabepos} *)
	ST_WT_Transport_Abgabe.e_wt_abgabepos_verlassen AT %IX28.3 : BOOL;	(*  ~ {LinkedWith:TIID^Gerät 1 (EtherCAT)^Schaltschrank (EK1100)^A32 (EL1819)^Channel 12^ST_WT_Transport_Abgabe.e_wt_abgabepos_verlassen} *)
	ST_WT_Transport_Achse.fb_axis.e_limit_sensor_positive AT %IX1447.0 : BOOL;
	ST_WT_Transport_Achse.fb_axis.e_limit_sensor_negative AT %IX1447.1 : BOOL;
	ST_WT_Transport_Achse.fb_axis.e_referenz_sensor AT %IX1447.2 : BOOL;
	ST_WT_Transport_Achse.e_referenz_sensor AT %IX1446.2 : BOOL;
	ST_WT_Transport_Achse.i16_torque AT %IB1444 : INT;
	ST_WT_Transport_Beladen.e_wt_auf_beladepos AT %IX28.4 : BOOL;	(*  ~ {LinkedWith:TIID^Gerät 1 (EtherCAT)^Schaltschrank (EK1100)^A32 (EL1819)^Channel 9^ST_WT_Transport_Beladen.e_wt_auf_beladepos} *)
	ST_WT_Transport_Beladen.e_wt_im_aktionsfeld AT %IX28.5 : BOOL;	(*  ~ {LinkedWith:TIID^Gerät 1 (EtherCAT)^Schaltschrank (EK1100)^A31 (EL1819)^Channel 8^ST_WT_Transport_Beladen.e_wt_im_aktionsfeld} *)
	ST_WT_Transport_Beladen.e_wt_beladepos_verlassen AT %IX28.6 : BOOL;	(*  ~ {LinkedWith:TIID^Gerät 1 (EtherCAT)^Schaltschrank (EK1100)^A32 (EL1819)^Channel 10^ST_WT_Transport_Beladen.e_wt_beladepos_verlassen} *)
	ST_WT_Transport_Beladen.e_wt_auf_pufferstrecke AT %IX28.7 : BOOL;	(*  ~ {LinkedWith:TIID^Gerät 1 (EtherCAT)^Schaltschrank (EK1100)^A32 (EL1819)^Channel 14^ST_WT_Transport_Beladen.e_wt_auf_pufferstrecke} *)
	ST_WT_Transport_Beladen.e_wt_faellt_in_achse_ueberw AT %IX880.5 : BOOL;	(*  ~ {LinkedWith:TIID^Gerät 1 (EtherCAT)^A37 Transportsystem (EP2338-0001)^Channel 7^ST_WT_Transport_Beladen.e_wt_faellt_in_achse_ueberw} *)
	ST_WT_Transport_Beladen_1720.e_wt_auf_beladepos AT %IX29.0 : BOOL;
	ST_WT_Transport_Beladen_1720.e_wt_im_aktionsfeld AT %IX29.1 : BOOL;
	ST_WT_Transport_Beladen_1720.e_wt_beladepos_verlassen AT %IX29.2 : BOOL;
	ST_WT_Transport_Beladen_1720.e_wt_auf_pufferstrecke AT %IX29.3 : BOOL;
	ST_WT_Transport_Beladen_Achse_1700.e_wt_auf_beladepos AT %IX1446.3 : BOOL;
	ST_WT_Transport_Beladen_Achse_1700.e_wt_beladepos_verlassen AT %IX1446.4 : BOOL;
	ST_WT_Transport_Beladen_Achse_1700.e_wt_auf_pufferstrecke AT %IX1446.5 : BOOL;
	ST_WT_Transport_Kontroller.e_stausensor_wt_ruecktransport AT %IX29.4 : BOOL;	(*  ~ {LinkedWith:TIID^Gerät 1 (EtherCAT)^Schaltschrank (EK1100)^A32 (EL1819)^Channel 13^ST_WT_Transport_Kontroller.e_stausensor_wt_ruecktransport} *)
	ST_WT_Transport_Kontroller.a_foerderband_wt_transport AT %QX8.5 : BOOL;	(*  ~ {LinkedWith:TIID^Gerät 1 (EtherCAT)^Schaltschrank (EK1100)^A46 (EL2809)^Channel 8^ST_WT_Transport_Kontroller.a_foerderband_wt_transport} *)
	ST_WT_Transport_Kontroller.a_foerderband_wt_ruecktransport AT %QX8.6 : BOOL;	(*  ~ {LinkedWith:TIID^Gerät 1 (EtherCAT)^Schaltschrank (EK1100)^A46 (EL2809)^Channel 13^ST_WT_Transport_Kontroller.a_foerderband_wt_ruecktransport} *)
	ST_WT_Transport_Kontroller.e_ueberstrom_foerderbaender AT %IX1580.0 : BOOL;
	ST_WT_Transport_Warteposition_1700.e_wt_auf_wartepos_1700 AT %IX1446.6 : BOOL;
	ST_WT_Transport_Warteposition_1700.e_wt_wartepos_verlassen_1700 AT %IX1446.7 : BOOL;
	ST_WT_Transport_Warteposition_1720.e_wt_auf_wartepos AT %IX29.5 : BOOL;
	ST_WT_Transport_Warteposition_1720.e_wt_wartepos_verlassen AT %IX29.6 : BOOL;
	ST_Y_Achse.fb_axis.e_limit_sensor_positive AT %IX31.3 : BOOL;
	ST_Y_Achse.fb_axis.e_limit_sensor_negative AT %IX31.4 : BOOL;
	ST_Y_Achse.fb_axis.e_referenz_sensor AT %IX31.5 : BOOL;
	ST_Y_Achse.e_referenz_sensor AT %IX29.7 : BOOL;
	ST_Y_Achse.i16_torque AT %IB4 : INT;
	ST_Y_Achse.i16_DigitalInput AT %IB1276 : INT;	(*  ~ {LinkedWith:TIID^Gerät 1 (EtherCAT)^A6 YZ-Achse (AX5201-0000-0011)^AT 1^Digital inputs, state} *)
	ST_Z_Achse.fb_axis.e_limit_sensor_positive AT %IX32.1 : BOOL;
	ST_Z_Achse.fb_axis.e_limit_sensor_negative AT %IX32.2 : BOOL;
	ST_Z_Achse.fb_axis.e_referenz_sensor AT %IX32.3 : BOOL;
	ST_Z_Achse.e_referenz_sensor AT %IX30.0 : BOOL;
	ST_Z_Achse.i16_torque AT %IB6 : INT;
	ST_Z_Achse.i16_DigitalInput AT %IB1278 : INT;	(*  ~ {LinkedWith:TIID^Gerät 1 (EtherCAT)^A6 YZ-Achse (AX5201-0000-0011)^AT 1^Digital inputs, state} *)
	ST_Z_Achse.e_kontrolle_rastnase AT %IX1280.7 : BOOL;
	.z_achse.PlcToNc AT %QB10 : PLCTONC_AXIS_REF;	(*  ~ {LinkedWith:TINC^NC-Task 1 SAF^Achsen^Z_Achse^Eingänge^.z_achse.PlcToNc} *)
	.z_achse.NcToPlc AT %IB33 : NCTOPLC_AXIS_REF;	(*  ~ {LinkedWith:TINC^NC-Task 1 SAF^Achsen^Z_Achse^Ausgänge^.z_achse.NcToPlc} *)
	.bestueckachse.PlcToNc AT %QB138 : PLCTONC_AXIS_REF;	(*  ~ {LinkedWith:TINC^NC-Task 1 SAF^Achsen^Bestueckachse^Eingänge^.bestueckachse.PlcToNc} *)
	.bestueckachse.NcToPlc AT %IB161 : NCTOPLC_AXIS_REF;	(*  ~ {LinkedWith:TINC^NC-Task 1 SAF^Achsen^Bestueckachse^Ausgänge^Bestueckachse_ToPlc} *)
	.virtuelle_master_achse.PlcToNc AT %QB754 : PLCTONC_AXIS_REF;	(*  ~ {LinkedWith:TINC^NC-Task 1 SAF^Achsen^Virtuelle_Masterachse^Eingänge^.virtuelle_master_achse.PlcToNc} *)
	.virtuelle_master_achse.NcToPlc AT %IB882 : NCTOPLC_AXIS_REF;	(*  ~ {LinkedWith:TINC^NC-Task 1 SAF^Achsen^Virtuelle_Masterachse^Ausgänge^.virtuelle_master_achse.NcToPlc} *)
	.getriebe_einstell_achse.PlcToNc AT %QB882 : PLCTONC_AXIS_REF;
	.getriebe_einstell_achse.NcToPlc AT %IB1010 : NCTOPLC_AXIS_REF;	(*  ~ {LinkedWith:TINC^NC-Task 1 SAF^Achsen^Getriebe_Einstellachse^Ausgänge^.getriebe_einstell_achse.NcToPlc} *)
	.y_achse.PlcToNc AT %QB394 : PLCTONC_AXIS_REF;	(*  ~ {LinkedWith:TINC^NC-Task 1 SAF^Achsen^Y_Achse^Eingänge^.y_achse.PlcToNc} *)
	.y_achse.NcToPlc AT %IB417 : NCTOPLC_AXIS_REF;	(*  ~ {LinkedWith:TINC^NC-Task 1 SAF^Achsen^Y_Achse^Ausgänge^.y_achse.NcToPlc} *)
	.b_achse.PlcToNc AT %QB1010 : PLCTONC_AXIS_REF;
	.b_achse.NcToPlc AT %IB1138 : NCTOPLC_AXIS_REF;
	.transport_wt_achse.PlcToNc AT %QB1309 : PLCTONC_AXIS_REF;
	.transport_wt_achse.NcToPlc AT %IB1448 : NCTOPLC_AXIS_REF;
	.e_smema_station_vorher_in_anforderung AT %IX30.1 : BOOL;	(*  ~ {LinkedWith:TIID^Gerät 1 (EtherCAT)^Schaltschrank (EK1100)^A31 (EL1819)^Channel 7^e_smema_station_vorher_in_anforderung} *)
	.e_smema_station_vorher_in_abgegeben AT %IX30.2 : BOOL;	(*  ~ {LinkedWith:TIID^Gerät 1 (EtherCAT)^Schaltschrank (EK1100)^A31 (EL1819)^Channel 6^e_smema_station_vorher_in_abgegeben} *)
	.a_smema_station_vorher_out_erlaubnis AT %QX9.0 : BOOL;	(*  ~ {LinkedWith:TIID^Gerät 1 (EtherCAT)^Schaltschrank (EK1100)^A47 (EL2809)^Channel 10^a_smema_station_vorher_out_erlaubnis} *)
	.a_smema_station_vorher_out_angekommen AT %QX9.1 : BOOL;	(*  ~ {LinkedWith:TIID^Gerät 1 (EtherCAT)^Schaltschrank (EK1100)^A47 (EL2809)^Channel 9^a_smema_station_vorher_out_angekommen} *)
	.e_smema_station_nachher_in_erlaubnis AT %IX30.3 : BOOL;	(*  ~ {LinkedWith:TIID^Gerät 1 (EtherCAT)^Schaltschrank (EK1100)^A31 (EL1819)^Channel 13^e_smema_station_nachher_in_erlaubnis} *)
	.e_smema_station_nachher_in_angekommen AT %IX30.4 : BOOL;	(*  ~ {LinkedWith:TIID^Gerät 1 (EtherCAT)^Schaltschrank (EK1100)^A31 (EL1819)^Channel 12^e_smema_station_nachher_in_angekommen} *)
	.a_smema_station_nachher_out_anforderung AT %QX9.2 : BOOL;	(*  ~ {LinkedWith:TIID^Gerät 1 (EtherCAT)^Schaltschrank (EK1100)^A47 (EL2809)^Channel 12^a_smema_station_nachher_out_anforderung} *)
	.a_smema_station_nachher_out_abgegeben AT %QX9.3 : BOOL;	(*  ~ {LinkedWith:TIID^Gerät 1 (EtherCAT)^Schaltschrank (EK1100)^A47 (EL2809)^Channel 11^a_smema_station_nachher_out_abgegeben} *)
	.a_zyl_vorschub_einfahren AT %QX9.4 : BOOL;	(*  ~ {LinkedWith:TIID^Gerät 1 (EtherCAT)^A50 (CPX-FB38 64Byte)^Outputs^QB4^a_zyl_vorschub_einfahren} *)
	.a_zyl_vorschub_ausfahren AT %QX9.5 : BOOL;	(*  ~ {LinkedWith:TIID^Gerät 1 (EtherCAT)^A50 (CPX-FB38 64Byte)^Outputs^QB4^a_zyl_vorschub_ausfahren} *)
	.a_zyl_faenger_einfahren AT %QX9.6 : BOOL;	(*  ~ {LinkedWith:TIID^Gerät 1 (EtherCAT)^A150 (EP2338-0001)^Channel 7^a_zyl_faenger_einfahren} *)
	.a_zyl_klemmen_einfahren AT %QX9.7 : BOOL;	(*  ~ {LinkedWith:TIID^Gerät 1 (EtherCAT)^A150 (EP2338-0001)^Channel 8^a_zyl_klemmen_einfahren} *)
	.haspel_re.fb.e_haspel_notaus AT %IX673.0 : BOOL;	(*  ~ {LinkedWith:TIID^Gerät 1 (EtherCAT)^A36 Haspel 2 - Rechts (EP2338-0001)^Channel 7^.haspel_re.fb.e_haspel_notaus} *)
	.haspel_re.fb.e_haspel_bandende AT %IX673.1 : BOOL;	(*  ~ {LinkedWith:TIID^Gerät 1 (EtherCAT)^A36 Haspel 2 - Rechts (EP2338-0001)^Channel 8^.haspel_re.fb.e_haspel_bandende} *)
	.haspel_re.fb.e_haspel_einschalten AT %IX673.2 : BOOL;	(*  ~ {LinkedWith:TIID^Gerät 1 (EtherCAT)^A36 Haspel 2 - Rechts (EP2338-0001)^Channel 5^.haspel_re.fb.e_haspel_einschalten} *)
	.haspel_re.fb.e_haspel_ausschalten AT %IX673.3 : BOOL;	(*  ~ {LinkedWith:TIID^Gerät 1 (EtherCAT)^A36 Haspel 2 - Rechts (EP2338-0001)^Channel 6^.haspel_re.fb.e_haspel_ausschalten} *)
	.haspel_li.fb.e_haspel_notaus AT %IX673.4 : BOOL;	(*  ~ {LinkedWith:TIID^Gerät 1 (EtherCAT)^A35 Haspel 1 - Links (EP2338-0001)^Channel 7^.haspel_li.fb.e_haspel_notaus} *)
	.haspel_li.fb.e_haspel_bandende AT %IX673.5 : BOOL;	(*  ~ {LinkedWith:TIID^Gerät 1 (EtherCAT)^A35 Haspel 1 - Links (EP2338-0001)^Channel 8^.haspel_li.fb.e_haspel_bandende} *)
	.haspel_li.fb.e_haspel_einschalten AT %IX673.6 : BOOL;	(*  ~ {LinkedWith:TIID^Gerät 1 (EtherCAT)^A35 Haspel 1 - Links (EP2338-0001)^Channel 5^.haspel_li.fb.e_haspel_einschalten} *)
	.haspel_li.fb.e_haspel_ausschalten AT %IX673.7 : BOOL;	(*  ~ {LinkedWith:TIID^Gerät 1 (EtherCAT)^A35 Haspel 1 - Links (EP2338-0001)^Channel 6^.haspel_li.fb.e_haspel_ausschalten} *)
	.betriebsstundenzaehler.fb.a_betriebsstundenzaehler AT %QX650.0 : BOOL;	(*  ~ {LinkedWith:TIID^Gerät 1 (EtherCAT)^Schaltschrank (EK1100)^A46 (EL2809)^Channel 15^.betriebsstundenzaehler.fb.a_betriebsstundenzaehler} *)
	.balluff_tag_reader.fb.EL6ComInData AT %IB674 : EL6inData22B;	(*  ~ {LinkedWith:TIID^Gerät 1 (EtherCAT)^Schaltschrank (EK1100)^A40 (EL6001)^COM Inputs^Status;
																				TIID^Gerät 1 (EtherCAT)^Schaltschrank (EK1100)^A40 (EL6001)^COM Inputs^Data In 0;
																				TIID^Gerät 1 (EtherCAT)^Schaltschrank (EK1100)^A40 (EL6001)^COM Inputs^Data In 1;
																				TIID^Gerät 1 (EtherCAT)^Schaltschrank (EK1100)^A40 (EL6001)^COM Inputs^Data In 2;
																				TIID^Gerät 1 (EtherCAT)^Schaltschrank (EK1100)^A40 (EL6001)^COM Inputs^Data In 3;
																				TIID^Gerät 1 (EtherCAT)^Schaltschrank (EK1100)^A40 (EL6001)^COM Inputs^Data In 4;
																				TIID^Gerät 1 (EtherCAT)^Schaltschrank (EK1100)^A40 (EL6001)^COM Inputs^Data In 5;
																				TIID^Gerät 1 (EtherCAT)^Schaltschrank (EK1100)^A40 (EL6001)^COM Inputs^Data In 6;
																				TIID^Gerät 1 (EtherCAT)^Schaltschrank (EK1100)^A40 (EL6001)^COM Inputs^Data In 7;
																				TIID^Gerät 1 (EtherCAT)^Schaltschrank (EK1100)^A40 (EL6001)^COM Inputs^Data In 8;
																				TIID^Gerät 1 (EtherCAT)^Schaltschrank (EK1100)^A40 (EL6001)^COM Inputs^Data In 9;
																				TIID^Gerät 1 (EtherCAT)^Schaltschrank (EK1100)^A40 (EL6001)^COM Inputs^Data In 10;
																				TIID^Gerät 1 (EtherCAT)^Schaltschrank (EK1100)^A40 (EL6001)^COM Inputs^Data In 11;
																				TIID^Gerät 1 (EtherCAT)^Schaltschrank (EK1100)^A40 (EL6001)^COM Inputs^Data In 12;
																				TIID^Gerät 1 (EtherCAT)^Schaltschrank (EK1100)^A40 (EL6001)^COM Inputs^Data In 13;
																				TIID^Gerät 1 (EtherCAT)^Schaltschrank (EK1100)^A40 (EL6001)^COM Inputs^Data In 14;
																				TIID^Gerät 1 (EtherCAT)^Schaltschrank (EK1100)^A40 (EL6001)^COM Inputs^Data In 15;
																				TIID^Gerät 1 (EtherCAT)^Schaltschrank (EK1100)^A40 (EL6001)^COM Inputs^Data In 16;
																				TIID^Gerät 1 (EtherCAT)^Schaltschrank (EK1100)^A40 (EL6001)^COM Inputs^Data In 17;
																				TIID^Gerät 1 (EtherCAT)^Schaltschrank (EK1100)^A40 (EL6001)^COM Inputs^Data In 18;
																				TIID^Gerät 1 (EtherCAT)^Schaltschrank (EK1100)^A40 (EL6001)^COM Inputs^Data In 19;
																				TIID^Gerät 1 (EtherCAT)^Schaltschrank (EK1100)^A40 (EL6001)^COM Inputs^Data In 20;
																				TIID^Gerät 1 (EtherCAT)^Schaltschrank (EK1100)^A40 (EL6001)^COM Inputs^Data In 21} *)
	.balluff_tag_reader.fb.EL6ComOutData AT %QB651 : EL6outData22B;	(*  ~ {LinkedWith:TIID^Gerät 1 (EtherCAT)^Schaltschrank (EK1100)^A40 (EL6001)^COM Outputs^Ctrl;
																					TIID^Gerät 1 (EtherCAT)^Schaltschrank (EK1100)^A40 (EL6001)^COM Outputs^Data Out 0;
																					TIID^Gerät 1 (EtherCAT)^Schaltschrank (EK1100)^A40 (EL6001)^COM Outputs^Data Out 1;
																					TIID^Gerät 1 (EtherCAT)^Schaltschrank (EK1100)^A40 (EL6001)^COM Outputs^Data Out 2;
																					TIID^Gerät 1 (EtherCAT)^Schaltschrank (EK1100)^A40 (EL6001)^COM Outputs^Data Out 3;
																					TIID^Gerät 1 (EtherCAT)^Schaltschrank (EK1100)^A40 (EL6001)^COM Outputs^Data Out 4;
																					TIID^Gerät 1 (EtherCAT)^Schaltschrank (EK1100)^A40 (EL6001)^COM Outputs^Data Out 5;
																					TIID^Gerät 1 (EtherCAT)^Schaltschrank (EK1100)^A40 (EL6001)^COM Outputs^Data Out 6;
																					TIID^Gerät 1 (EtherCAT)^Schaltschrank (EK1100)^A40 (EL6001)^COM Outputs^Data Out 7;
																					TIID^Gerät 1 (EtherCAT)^Schaltschrank (EK1100)^A40 (EL6001)^COM Outputs^Data Out 8;
																					TIID^Gerät 1 (EtherCAT)^Schaltschrank (EK1100)^A40 (EL6001)^COM Outputs^Data Out 9;
																					TIID^Gerät 1 (EtherCAT)^Schaltschrank (EK1100)^A40 (EL6001)^COM Outputs^Data Out 10;
																					TIID^Gerät 1 (EtherCAT)^Schaltschrank (EK1100)^A40 (EL6001)^COM Outputs^Data Out 11;
																					TIID^Gerät 1 (EtherCAT)^Schaltschrank (EK1100)^A40 (EL6001)^COM Outputs^Data Out 12;
																					TIID^Gerät 1 (EtherCAT)^Schaltschrank (EK1100)^A40 (EL6001)^COM Outputs^Data Out 13;
																					TIID^Gerät 1 (EtherCAT)^Schaltschrank (EK1100)^A40 (EL6001)^COM Outputs^Data Out 14;
																					TIID^Gerät 1 (EtherCAT)^Schaltschrank (EK1100)^A40 (EL6001)^COM Outputs^Data Out 15;
																					TIID^Gerät 1 (EtherCAT)^Schaltschrank (EK1100)^A40 (EL6001)^COM Outputs^Data Out 16;
																					TIID^Gerät 1 (EtherCAT)^Schaltschrank (EK1100)^A40 (EL6001)^COM Outputs^Data Out 17;
																					TIID^Gerät 1 (EtherCAT)^Schaltschrank (EK1100)^A40 (EL6001)^COM Outputs^Data Out 18;
																					TIID^Gerät 1 (EtherCAT)^Schaltschrank (EK1100)^A40 (EL6001)^COM Outputs^Data Out 19;
																					TIID^Gerät 1 (EtherCAT)^Schaltschrank (EK1100)^A40 (EL6001)^COM Outputs^Data Out 20;
																					TIID^Gerät 1 (EtherCAT)^Schaltschrank (EK1100)^A40 (EL6001)^COM Outputs^Data Out 21} *)
	.balluff_tag_reader.fb.e_tag_im_aktionsfeld AT %IX698.0 : BOOL;	(*  ~ {LinkedWith:TIID^Gerät 1 (EtherCAT)^Schaltschrank (EK1100)^A31 (EL1819)^Channel 8^ST_WT_Transport_Beladen.e_wt_im_aktionsfeld} *)
	.barcode.fb.COM_in_data AT %IB699 : PcComInData;	(*  ~ {LinkedWith:TIID^Gerät 4 (COM Port)^Eingänge^SerStatus;
																	TIID^Gerät 4 (COM Port)^Eingänge^Data1;
																	TIID^Gerät 4 (COM Port)^Eingänge^Data2;
																	TIID^Gerät 4 (COM Port)^Eingänge^Data3;
																	TIID^Gerät 4 (COM Port)^Eingänge^Data4;
																	TIID^Gerät 4 (COM Port)^Eingänge^Data5;
																	TIID^Gerät 4 (COM Port)^Eingänge^Data6;
																	TIID^Gerät 4 (COM Port)^Eingänge^Data7;
																	TIID^Gerät 4 (COM Port)^Eingänge^Data8;
																	TIID^Gerät 4 (COM Port)^Eingänge^Data9;
																	TIID^Gerät 4 (COM Port)^Eingänge^Data10;
																	TIID^Gerät 4 (COM Port)^Eingänge^Data11;
																	TIID^Gerät 4 (COM Port)^Eingänge^Data12;
																	TIID^Gerät 4 (COM Port)^Eingänge^Data13;
																	TIID^Gerät 4 (COM Port)^Eingänge^Data14;
																	TIID^Gerät 4 (COM Port)^Eingänge^Data15;
																	TIID^Gerät 4 (COM Port)^Eingänge^Data16;
																	TIID^Gerät 4 (COM Port)^Eingänge^Data17;
																	TIID^Gerät 4 (COM Port)^Eingänge^Data18;
																	TIID^Gerät 4 (COM Port)^Eingänge^Data19;
																	TIID^Gerät 4 (COM Port)^Eingänge^Data20;
																	TIID^Gerät 4 (COM Port)^Eingänge^Data21;
																	TIID^Gerät 4 (COM Port)^Eingänge^Data22;
																	TIID^Gerät 4 (COM Port)^Eingänge^Data23;
																	TIID^Gerät 4 (COM Port)^Eingänge^Data24;
																	TIID^Gerät 4 (COM Port)^Eingänge^Data25;
																	TIID^Gerät 4 (COM Port)^Eingänge^Data26;
																	TIID^Gerät 4 (COM Port)^Eingänge^Data27;
																	TIID^Gerät 4 (COM Port)^Eingänge^Data28;
																	TIID^Gerät 4 (COM Port)^Eingänge^Data29;
																	TIID^Gerät 4 (COM Port)^Eingänge^Data30;
																	TIID^Gerät 4 (COM Port)^Eingänge^Data31;
																	TIID^Gerät 4 (COM Port)^Eingänge^Data32;
																	TIID^Gerät 4 (COM Port)^Eingänge^Data33;
																	TIID^Gerät 4 (COM Port)^Eingänge^Data34;
																	TIID^Gerät 4 (COM Port)^Eingänge^Data35;
																	TIID^Gerät 4 (COM Port)^Eingänge^Data36;
																	TIID^Gerät 4 (COM Port)^Eingänge^Data37;
																	TIID^Gerät 4 (COM Port)^Eingänge^Data38;
																	TIID^Gerät 4 (COM Port)^Eingänge^Data39;
																	TIID^Gerät 4 (COM Port)^Eingänge^Data40;
																	TIID^Gerät 4 (COM Port)^Eingänge^Data41;
																	TIID^Gerät 4 (COM Port)^Eingänge^Data42;
																	TIID^Gerät 4 (COM Port)^Eingänge^Data43;
																	TIID^Gerät 4 (COM Port)^Eingänge^Data44;
																	TIID^Gerät 4 (COM Port)^Eingänge^Data45;
																	TIID^Gerät 4 (COM Port)^Eingänge^Data46;
																	TIID^Gerät 4 (COM Port)^Eingänge^Data47;
																	TIID^Gerät 4 (COM Port)^Eingänge^Data48;
																	TIID^Gerät 4 (COM Port)^Eingänge^Data49;
																	TIID^Gerät 4 (COM Port)^Eingänge^Data50;
																	TIID^Gerät 4 (COM Port)^Eingänge^Data51;
																	TIID^Gerät 4 (COM Port)^Eingänge^Data52;
																	TIID^Gerät 4 (COM Port)^Eingänge^Data53;
																	TIID^Gerät 4 (COM Port)^Eingänge^Data54;
																	TIID^Gerät 4 (COM Port)^Eingänge^Data55;
																	TIID^Gerät 4 (COM Port)^Eingänge^Data56;
																	TIID^Gerät 4 (COM Port)^Eingänge^Data57;
																	TIID^Gerät 4 (COM Port)^Eingänge^Data58;
																	TIID^Gerät 4 (COM Port)^Eingänge^Data59;
																	TIID^Gerät 4 (COM Port)^Eingänge^Data60;
																	TIID^Gerät 4 (COM Port)^Eingänge^Data61;
																	TIID^Gerät 4 (COM Port)^Eingänge^Data62;
																	TIID^Gerät 4 (COM Port)^Eingänge^Data63;
																	TIID^Gerät 4 (COM Port)^Eingänge^Data64} *)
	.barcode.fb.COM_out_data AT %QB675 : PcComOutData;	(*  ~ {LinkedWith:TIID^Gerät 4 (COM Port)^Ausgänge^SerCtrl;
																		TIID^Gerät 4 (COM Port)^Ausgänge^Data1;
																		TIID^Gerät 4 (COM Port)^Ausgänge^Data2;
																		TIID^Gerät 4 (COM Port)^Ausgänge^Data3;
																		TIID^Gerät 4 (COM Port)^Ausgänge^Data4;
																		TIID^Gerät 4 (COM Port)^Ausgänge^Data5;
																		TIID^Gerät 4 (COM Port)^Ausgänge^Data6;
																		TIID^Gerät 4 (COM Port)^Ausgänge^Data7;
																		TIID^Gerät 4 (COM Port)^Ausgänge^Data8;
																		TIID^Gerät 4 (COM Port)^Ausgänge^Data9;
																		TIID^Gerät 4 (COM Port)^Ausgänge^Data10;
																		TIID^Gerät 4 (COM Port)^Ausgänge^Data11;
																		TIID^Gerät 4 (COM Port)^Ausgänge^Data12;
																		TIID^Gerät 4 (COM Port)^Ausgänge^Data13;
																		TIID^Gerät 4 (COM Port)^Ausgänge^Data14;
																		TIID^Gerät 4 (COM Port)^Ausgänge^Data15;
																		TIID^Gerät 4 (COM Port)^Ausgänge^Data16;
																		TIID^Gerät 4 (COM Port)^Ausgänge^Data17;
																		TIID^Gerät 4 (COM Port)^Ausgänge^Data18;
																		TIID^Gerät 4 (COM Port)^Ausgänge^Data19;
																		TIID^Gerät 4 (COM Port)^Ausgänge^Data20;
																		TIID^Gerät 4 (COM Port)^Ausgänge^Data21;
																		TIID^Gerät 4 (COM Port)^Ausgänge^Data22;
																		TIID^Gerät 4 (COM Port)^Ausgänge^Data23;
																		TIID^Gerät 4 (COM Port)^Ausgänge^Data24;
																		TIID^Gerät 4 (COM Port)^Ausgänge^Data25;
																		TIID^Gerät 4 (COM Port)^Ausgänge^Data26;
																		TIID^Gerät 4 (COM Port)^Ausgänge^Data27;
																		TIID^Gerät 4 (COM Port)^Ausgänge^Data28;
																		TIID^Gerät 4 (COM Port)^Ausgänge^Data29;
																		TIID^Gerät 4 (COM Port)^Ausgänge^Data30;
																		TIID^Gerät 4 (COM Port)^Ausgänge^Data31;
																		TIID^Gerät 4 (COM Port)^Ausgänge^Data32;
																		TIID^Gerät 4 (COM Port)^Ausgänge^Data33;
																		TIID^Gerät 4 (COM Port)^Ausgänge^Data34;
																		TIID^Gerät 4 (COM Port)^Ausgänge^Data35;
																		TIID^Gerät 4 (COM Port)^Ausgänge^Data36;
																		TIID^Gerät 4 (COM Port)^Ausgänge^Data37;
																		TIID^Gerät 4 (COM Port)^Ausgänge^Data38;
																		TIID^Gerät 4 (COM Port)^Ausgänge^Data39;
																		TIID^Gerät 4 (COM Port)^Ausgänge^Data40;
																		TIID^Gerät 4 (COM Port)^Ausgänge^Data41;
																		TIID^Gerät 4 (COM Port)^Ausgänge^Data42;
																		TIID^Gerät 4 (COM Port)^Ausgänge^Data43;
																		TIID^Gerät 4 (COM Port)^Ausgänge^Data44;
																		TIID^Gerät 4 (COM Port)^Ausgänge^Data45;
																		TIID^Gerät 4 (COM Port)^Ausgänge^Data46;
																		TIID^Gerät 4 (COM Port)^Ausgänge^Data47;
																		TIID^Gerät 4 (COM Port)^Ausgänge^Data48;
																		TIID^Gerät 4 (COM Port)^Ausgänge^Data49;
																		TIID^Gerät 4 (COM Port)^Ausgänge^Data50;
																		TIID^Gerät 4 (COM Port)^Ausgänge^Data51;
																		TIID^Gerät 4 (COM Port)^Ausgänge^Data52;
																		TIID^Gerät 4 (COM Port)^Ausgänge^Data53;
																		TIID^Gerät 4 (COM Port)^Ausgänge^Data54;
																		TIID^Gerät 4 (COM Port)^Ausgänge^Data55;
																		TIID^Gerät 4 (COM Port)^Ausgänge^Data56;
																		TIID^Gerät 4 (COM Port)^Ausgänge^Data57;
																		TIID^Gerät 4 (COM Port)^Ausgänge^Data58;
																		TIID^Gerät 4 (COM Port)^Ausgänge^Data59;
																		TIID^Gerät 4 (COM Port)^Ausgänge^Data60;
																		TIID^Gerät 4 (COM Port)^Ausgänge^Data61;
																		TIID^Gerät 4 (COM Port)^Ausgänge^Data62;
																		TIID^Gerät 4 (COM Port)^Ausgänge^Data63;
																		TIID^Gerät 4 (COM Port)^Ausgänge^Data64} *)
	.kraftmessdose.fb.st_sensor AT %IB766 : struct_analog_in;
	.EtherCatDiag[1].by_AmsNetId AT %IB1581 : T_AmsNetIdArr;
	.EtherCatDiag[2].by_AmsNetId AT %IB1587 : T_AmsNetIdArr;
	.EtherCatDiag[3].by_AmsNetId AT %IB1593 : T_AmsNetIdArr;
	.EtherCatDiag[4].by_AmsNetId AT %IB1599 : T_AmsNetIdArr;
	.zyl_wt_zentrierer_tisch.fb.e_sensor1_eingefahren AT %IX773.0 : BOOL;	(*  ~ {LinkedWith:TIID^Gerät 1 (EtherCAT)^A37 Transportsystem (EP2338-0001)^Channel 3^.zyl_wt_zentrierer_tisch.fb.e_sensor1_eingefahren} *)
	.zyl_wt_zentrierer_tisch.fb.e_sensor1_ausgefahren AT %IX773.1 : BOOL;	(*  ~ {LinkedWith:TIID^Gerät 1 (EtherCAT)^A37 Transportsystem (EP2338-0001)^Channel 4^.zyl_wt_zentrierer_tisch.fb.e_sensor1_ausgefahren} *)
	.zyl_wt_zentrierer_tisch.fb.e_sensor2_eingefahren AT %IX773.2 : BOOL;	(*  ~ {LinkedWith:TIID^Gerät 1 (EtherCAT)^A37 Transportsystem (EP2338-0001)^Channel 5^.zyl_wt_zentrierer_tisch.fb.e_sensor2_eingefahren} *)
	.zyl_wt_zentrierer_tisch.fb.e_sensor2_ausgefahren AT %IX773.3 : BOOL;	(*  ~ {LinkedWith:TIID^Gerät 1 (EtherCAT)^A37 Transportsystem (EP2338-0001)^Channel 6^.zyl_wt_zentrierer_tisch.fb.e_sensor2_ausgefahren} *)
	.zyl_wt_zentrierer_tisch.fb.e_sensor3_eingefahren AT %IX773.4 : BOOL;
	.zyl_wt_zentrierer_tisch.fb.e_sensor3_ausgefahren AT %IX773.5 : BOOL;
	.zyl_wt_zentrierer_tisch.fb.e_sensor_mittegefahren AT %IX773.6 : BOOL;
	.zyl_wt_zentrierer_tisch.fb.e_taste_einfahren AT %IX773.7 : BOOL;
	.zyl_wt_zentrierer_tisch.fb.e_taste_ausfahren AT %IX774.0 : BOOL;
	.zyl_wt_zentrierer_tisch.fb.a_ventil_einfahren AT %QX741.1 : BOOL;	(*  ~ {LinkedWith:TIID^Gerät 1 (EtherCAT)^A50 (CPX-FB38 64Byte)^Outputs^QB0^.zyl_wt_zentrierer_tisch.fb.a_ventil_einfahren} *)
	.zyl_wt_zentrierer_tisch.fb.a_ventil_ausfahren AT %QX741.2 : BOOL;	(*  ~ {LinkedWith:TIID^Gerät 1 (EtherCAT)^A50 (CPX-FB38 64Byte)^Outputs^QB0^.zyl_wt_zentrierer_tisch.fb.a_ventil_ausfahren} *)
	.zyl_wt_stopper_tisch.fb.e_sensor1_eingefahren AT %IX774.1 : BOOL;	(*  ~ {LinkedWith:TIID^Gerät 1 (EtherCAT)^A37 Transportsystem (EP2338-0001)^Channel 1^.zyl_wt_stopper_tisch.fb.e_sensor1_eingefahren} *)
	.zyl_wt_stopper_tisch.fb.e_sensor1_ausgefahren AT %IX774.2 : BOOL;	(*  ~ {LinkedWith:TIID^Gerät 1 (EtherCAT)^A37 Transportsystem (EP2338-0001)^Channel 2^.zyl_wt_stopper_tisch.fb.e_sensor1_ausgefahren} *)
	.zyl_wt_stopper_tisch.fb.e_sensor2_eingefahren AT %IX774.3 : BOOL;
	.zyl_wt_stopper_tisch.fb.e_sensor2_ausgefahren AT %IX774.4 : BOOL;
	.zyl_wt_stopper_tisch.fb.e_sensor3_eingefahren AT %IX774.5 : BOOL;
	.zyl_wt_stopper_tisch.fb.e_sensor3_ausgefahren AT %IX774.6 : BOOL;
	.zyl_wt_stopper_tisch.fb.e_sensor_mittegefahren AT %IX774.7 : BOOL;
	.zyl_wt_stopper_tisch.fb.e_taste_einfahren AT %IX775.0 : BOOL;
	.zyl_wt_stopper_tisch.fb.e_taste_ausfahren AT %IX775.1 : BOOL;
	.zyl_wt_stopper_tisch.fb.a_ventil_einfahren AT %QX741.3 : BOOL;	(*  ~ {LinkedWith:TIID^Gerät 1 (EtherCAT)^A50 (CPX-FB38 64Byte)^Outputs^QB0^.zyl_wt_stopper_tisch.fb.a_ventil_einfahren} *)
	.zyl_wt_stopper_tisch.fb.a_ventil_ausfahren AT %QX741.4 : BOOL;	(*  ~ {LinkedWith:TIID^Gerät 1 (EtherCAT)^A50 (CPX-FB38 64Byte)^Outputs^QB0^.zyl_wt_stopper_tisch.fb.a_ventil_ausfahren} *)
	.zyl_wt_stopper_auslauf.fb.e_sensor1_eingefahren AT %IX775.2 : BOOL;
	.zyl_wt_stopper_auslauf.fb.e_sensor1_ausgefahren AT %IX775.3 : BOOL;
	.zyl_wt_stopper_auslauf.fb.e_sensor2_eingefahren AT %IX775.4 : BOOL;
	.zyl_wt_stopper_auslauf.fb.e_sensor2_ausgefahren AT %IX775.5 : BOOL;
	.zyl_wt_stopper_auslauf.fb.e_sensor3_eingefahren AT %IX775.6 : BOOL;
	.zyl_wt_stopper_auslauf.fb.e_sensor3_ausgefahren AT %IX775.7 : BOOL;
	.zyl_wt_stopper_auslauf.fb.e_sensor_mittegefahren AT %IX776.0 : BOOL;
	.zyl_wt_stopper_auslauf.fb.e_taste_einfahren AT %IX776.1 : BOOL;
	.zyl_wt_stopper_auslauf.fb.e_taste_ausfahren AT %IX776.2 : BOOL;
	.zyl_wt_stopper_auslauf.fb.a_ventil_einfahren AT %QX741.5 : BOOL;	(*  ~ {LinkedWith:TIID^Gerät 1 (EtherCAT)^A50 (CPX-FB38 64Byte)^Outputs^QB1^.zyl_wt_stopper_auslauf.fb.a_ventil_einfahren} *)
	.zyl_wt_stopper_auslauf.fb.a_ventil_ausfahren AT %QX741.6 : BOOL;
	.zyl_haspel_re_heben.fb.e_sensor1_eingefahren AT %IX776.3 : BOOL;
	.zyl_haspel_re_heben.fb.e_sensor1_ausgefahren AT %IX776.4 : BOOL;	(*  ~ {LinkedWith:TIID^Gerät 1 (EtherCAT)^A36 Haspel 2 - Rechts (EP2338-0001)^Channel 2^.zyl_haspel_re_heben.fb.e_sensor1_ausgefahren} *)
	.zyl_haspel_re_heben.fb.e_sensor2_eingefahren AT %IX776.5 : BOOL;
	.zyl_haspel_re_heben.fb.e_sensor2_ausgefahren AT %IX776.6 : BOOL;
	.zyl_haspel_re_heben.fb.e_sensor3_eingefahren AT %IX776.7 : BOOL;
	.zyl_haspel_re_heben.fb.e_sensor3_ausgefahren AT %IX777.0 : BOOL;
	.zyl_haspel_re_heben.fb.e_sensor_mittegefahren AT %IX777.1 : BOOL;
	.zyl_haspel_re_heben.fb.e_taste_einfahren AT %IX777.2 : BOOL;
	.zyl_haspel_re_heben.fb.e_taste_ausfahren AT %IX777.3 : BOOL;
	.zyl_haspel_re_heben.fb.a_ventil_einfahren AT %QX741.7 : BOOL;	(*  ~ {LinkedWith:TIID^Gerät 1 (EtherCAT)^A50 (CPX-FB38 64Byte)^Outputs^QB2^.zyl_haspel_re_heben.fb.a_ventil_einfahren} *)
	.zyl_haspel_re_heben.fb.a_ventil_ausfahren AT %QX742.0 : BOOL;	(*  ~ {LinkedWith:TIID^Gerät 1 (EtherCAT)^A50 (CPX-FB38 64Byte)^Outputs^QB2^.zyl_haspel_re_heben.fb.a_ventil_ausfahren} *)
	.zyl_haspel_re_abspulen.fb.e_sensor1_eingefahren AT %IX777.4 : BOOL;
	.zyl_haspel_re_abspulen.fb.e_sensor1_ausgefahren AT %IX777.5 : BOOL;	(*  ~ {LinkedWith:TIID^Gerät 1 (EtherCAT)^A36 Haspel 2 - Rechts (EP2338-0001)^Channel 1^.zyl_haspel_re_abspulen.fb.e_sensor1_ausgefahren} *)
	.zyl_haspel_re_abspulen.fb.e_sensor2_eingefahren AT %IX777.6 : BOOL;
	.zyl_haspel_re_abspulen.fb.e_sensor2_ausgefahren AT %IX777.7 : BOOL;
	.zyl_haspel_re_abspulen.fb.e_sensor3_eingefahren AT %IX778.0 : BOOL;
	.zyl_haspel_re_abspulen.fb.e_sensor3_ausgefahren AT %IX778.1 : BOOL;
	.zyl_haspel_re_abspulen.fb.e_sensor_mittegefahren AT %IX778.2 : BOOL;
	.zyl_haspel_re_abspulen.fb.e_taste_einfahren AT %IX778.3 : BOOL;
	.zyl_haspel_re_abspulen.fb.e_taste_ausfahren AT %IX778.4 : BOOL;
	.zyl_haspel_re_abspulen.fb.a_ventil_einfahren AT %QX742.1 : BOOL;	(*  ~ {LinkedWith:TIID^Gerät 1 (EtherCAT)^A50 (CPX-FB38 64Byte)^Outputs^QB4^.zyl_haspel_re_abspulen.fb.a_ventil_einfahren} *)
	.zyl_haspel_re_abspulen.fb.a_ventil_ausfahren AT %QX742.2 : BOOL;	(*  ~ {LinkedWith:TIID^Gerät 1 (EtherCAT)^A50 (CPX-FB38 64Byte)^Outputs^QB4^.zyl_haspel_re_abspulen.fb.a_ventil_ausfahren} *)
	.zyl_haspel_li_heben.fb.e_sensor1_eingefahren AT %IX778.5 : BOOL;
	.zyl_haspel_li_heben.fb.e_sensor1_ausgefahren AT %IX778.6 : BOOL;	(*  ~ {LinkedWith:TIID^Gerät 1 (EtherCAT)^A35 Haspel 1 - Links (EP2338-0001)^Channel 2^.zyl_haspel_li_heben.fb.e_sensor1_ausgefahren} *)
	.zyl_haspel_li_heben.fb.e_sensor2_eingefahren AT %IX778.7 : BOOL;
	.zyl_haspel_li_heben.fb.e_sensor2_ausgefahren AT %IX779.0 : BOOL;
	.zyl_haspel_li_heben.fb.e_sensor3_eingefahren AT %IX779.1 : BOOL;
	.zyl_haspel_li_heben.fb.e_sensor3_ausgefahren AT %IX779.2 : BOOL;
	.zyl_haspel_li_heben.fb.e_sensor_mittegefahren AT %IX779.3 : BOOL;
	.zyl_haspel_li_heben.fb.e_taste_einfahren AT %IX779.4 : BOOL;
	.zyl_haspel_li_heben.fb.e_taste_ausfahren AT %IX779.5 : BOOL;
	.zyl_haspel_li_heben.fb.a_ventil_einfahren AT %QX742.3 : BOOL;	(*  ~ {LinkedWith:TIID^Gerät 1 (EtherCAT)^A50 (CPX-FB38 64Byte)^Outputs^QB2^.zyl_haspel_li_heben.fb.a_ventil_einfahren} *)
	.zyl_haspel_li_heben.fb.a_ventil_ausfahren AT %QX742.4 : BOOL;	(*  ~ {LinkedWith:TIID^Gerät 1 (EtherCAT)^A50 (CPX-FB38 64Byte)^Outputs^QB2^.zyl_haspel_li_heben.fb.a_ventil_ausfahren} *)
	.zyl_haspel_li_abspulen.fb.e_sensor1_eingefahren AT %IX779.6 : BOOL;
	.zyl_haspel_li_abspulen.fb.e_sensor1_ausgefahren AT %IX779.7 : BOOL;	(*  ~ {LinkedWith:TIID^Gerät 1 (EtherCAT)^A35 Haspel 1 - Links (EP2338-0001)^Channel 1^.zyl_haspel_li_abspulen.fb.e_sensor1_ausgefahren} *)
	.zyl_haspel_li_abspulen.fb.e_sensor2_eingefahren AT %IX780.0 : BOOL;
	.zyl_haspel_li_abspulen.fb.e_sensor2_ausgefahren AT %IX780.1 : BOOL;
	.zyl_haspel_li_abspulen.fb.e_sensor3_eingefahren AT %IX780.2 : BOOL;
	.zyl_haspel_li_abspulen.fb.e_sensor3_ausgefahren AT %IX780.3 : BOOL;
	.zyl_haspel_li_abspulen.fb.e_sensor_mittegefahren AT %IX780.4 : BOOL;
	.zyl_haspel_li_abspulen.fb.e_taste_einfahren AT %IX780.5 : BOOL;
	.zyl_haspel_li_abspulen.fb.e_taste_ausfahren AT %IX780.6 : BOOL;
	.zyl_haspel_li_abspulen.fb.a_ventil_einfahren AT %QX742.5 : BOOL;	(*  ~ {LinkedWith:TIID^Gerät 1 (EtherCAT)^A50 (CPX-FB38 64Byte)^Outputs^QB4^.zyl_haspel_li_abspulen.fb.a_ventil_einfahren} *)
	.zyl_haspel_li_abspulen.fb.a_ventil_ausfahren AT %QX742.6 : BOOL;	(*  ~ {LinkedWith:TIID^Gerät 1 (EtherCAT)^A50 (CPX-FB38 64Byte)^Outputs^QB4^.zyl_haspel_li_abspulen.fb.a_ventil_ausfahren} *)
	.zyl_haspel_re_sperren.fb.e_sensor1_eingefahren AT %IX780.7 : BOOL;	(*  ~ {LinkedWith:TIID^Gerät 1 (EtherCAT)^A36 Haspel 2 - Rechts (EP2338-0001)^Channel 3^.zyl_haspel_re_sperren.fb.e_sensor1_eingefahren} *)
	.zyl_haspel_re_sperren.fb.e_sensor1_ausgefahren AT %IX781.0 : BOOL;	(*  ~ {LinkedWith:TIID^Gerät 1 (EtherCAT)^A36 Haspel 2 - Rechts (EP2338-0001)^Channel 4^.zyl_haspel_re_sperren.fb.e_sensor1_ausgefahren} *)
	.zyl_haspel_re_sperren.fb.e_sensor2_eingefahren AT %IX781.1 : BOOL;
	.zyl_haspel_re_sperren.fb.e_sensor2_ausgefahren AT %IX781.2 : BOOL;
	.zyl_haspel_re_sperren.fb.e_sensor3_eingefahren AT %IX781.3 : BOOL;
	.zyl_haspel_re_sperren.fb.e_sensor3_ausgefahren AT %IX781.4 : BOOL;
	.zyl_haspel_re_sperren.fb.e_sensor_mittegefahren AT %IX781.5 : BOOL;
	.zyl_haspel_re_sperren.fb.e_taste_einfahren AT %IX781.6 : BOOL;
	.zyl_haspel_re_sperren.fb.e_taste_ausfahren AT %IX781.7 : BOOL;
	.zyl_haspel_re_sperren.fb.a_ventil_einfahren AT %QX742.7 : BOOL;	(*  ~ {LinkedWith:TIID^Gerät 1 (EtherCAT)^A50 (CPX-FB38 64Byte)^Outputs^QB2^.zyl_haspel_re_sperren.fb.a_ventil_einfahren} *)
	.zyl_haspel_re_sperren.fb.a_ventil_ausfahren AT %QX743.0 : BOOL;	(*  ~ {LinkedWith:TIID^Gerät 1 (EtherCAT)^A50 (CPX-FB38 64Byte)^Outputs^QB2^.zyl_haspel_re_sperren.fb.a_ventil_ausfahren} *)
	.zyl_haspel_li_sperren.fb.e_sensor1_eingefahren AT %IX782.0 : BOOL;	(*  ~ {LinkedWith:TIID^Gerät 1 (EtherCAT)^A35 Haspel 1 - Links (EP2338-0001)^Channel 3^.zyl_haspel_li_sperren.fb.e_sensor1_eingefahren} *)
	.zyl_haspel_li_sperren.fb.e_sensor1_ausgefahren AT %IX782.1 : BOOL;	(*  ~ {LinkedWith:TIID^Gerät 1 (EtherCAT)^A35 Haspel 1 - Links (EP2338-0001)^Channel 4^.zyl_haspel_li_sperren.fb.e_sensor1_ausgefahren} *)
	.zyl_haspel_li_sperren.fb.e_sensor2_eingefahren AT %IX782.2 : BOOL;
	.zyl_haspel_li_sperren.fb.e_sensor2_ausgefahren AT %IX782.3 : BOOL;
	.zyl_haspel_li_sperren.fb.e_sensor3_eingefahren AT %IX782.4 : BOOL;
	.zyl_haspel_li_sperren.fb.e_sensor3_ausgefahren AT %IX782.5 : BOOL;
	.zyl_haspel_li_sperren.fb.e_sensor_mittegefahren AT %IX782.6 : BOOL;
	.zyl_haspel_li_sperren.fb.e_taste_einfahren AT %IX782.7 : BOOL;
	.zyl_haspel_li_sperren.fb.e_taste_ausfahren AT %IX783.0 : BOOL;
	.zyl_haspel_li_sperren.fb.a_ventil_einfahren AT %QX743.1 : BOOL;	(*  ~ {LinkedWith:TIID^Gerät 1 (EtherCAT)^A50 (CPX-FB38 64Byte)^Outputs^QB2^.zyl_haspel_li_sperren.fb.a_ventil_einfahren} *)
	.zyl_haspel_li_sperren.fb.a_ventil_ausfahren AT %QX743.2 : BOOL;	(*  ~ {LinkedWith:TIID^Gerät 1 (EtherCAT)^A50 (CPX-FB38 64Byte)^Outputs^QB2^.zyl_haspel_li_sperren.fb.a_ventil_ausfahren} *)
	.zyl_hublift_rechts_lift.fb.e_sensor1_eingefahren AT %IX783.1 : BOOL;	(*  ~ {LinkedWith:TIID^Gerät 1 (EtherCAT)^A250 Hublift Rechts (EK1101)^A251 (EL1819)^Channel 1^.zyl_hublift_rechts_lift.fb.e_sensor1_eingefahren} *)
	.zyl_hublift_rechts_lift.fb.e_sensor1_ausgefahren AT %IX783.2 : BOOL;	(*  ~ {LinkedWith:TIID^Gerät 1 (EtherCAT)^A250 Hublift Rechts (EK1101)^A251 (EL1819)^Channel 2^.zyl_hublift_rechts_lift.fb.e_sensor1_ausgefahren} *)
	.zyl_hublift_rechts_lift.fb.e_sensor2_eingefahren AT %IX783.3 : BOOL;
	.zyl_hublift_rechts_lift.fb.e_sensor2_ausgefahren AT %IX783.4 : BOOL;
	.zyl_hublift_rechts_lift.fb.e_sensor3_eingefahren AT %IX783.5 : BOOL;
	.zyl_hublift_rechts_lift.fb.e_sensor3_ausgefahren AT %IX783.6 : BOOL;
	.zyl_hublift_rechts_lift.fb.e_sensor_mittegefahren AT %IX783.7 : BOOL;
	.zyl_hublift_rechts_lift.fb.e_taste_einfahren AT %IX784.0 : BOOL;
	.zyl_hublift_rechts_lift.fb.e_taste_ausfahren AT %IX784.1 : BOOL;
	.zyl_hublift_rechts_lift.fb.a_ventil_einfahren AT %QX743.3 : BOOL;	(*  ~ {LinkedWith:TIID^Gerät 1 (EtherCAT)^A250 Hublift Rechts (EK1101)^A253 (EL2809)^Channel 1^.zyl_hublift_rechts_lift.fb.a_ventil_einfahren} *)
	.zyl_hublift_rechts_lift.fb.a_ventil_ausfahren AT %QX743.4 : BOOL;	(*  ~ {LinkedWith:TIID^Gerät 1 (EtherCAT)^A250 Hublift Rechts (EK1101)^A253 (EL2809)^Channel 2^.zyl_hublift_rechts_lift.fb.a_ventil_ausfahren} *)
	.zyl_hublift_rechts_wt_einzug.fb.e_sensor1_eingefahren AT %IX784.2 : BOOL;	(*  ~ {LinkedWith:TIID^Gerät 1 (EtherCAT)^A250 Hublift Rechts (EK1101)^A251 (EL1819)^Channel 3^.zyl_hublift_rechts_wt_einzug.fb.e_sensor1_eingefahren} *)
	.zyl_hublift_rechts_wt_einzug.fb.e_sensor1_ausgefahren AT %IX784.3 : BOOL;	(*  ~ {LinkedWith:TIID^Gerät 1 (EtherCAT)^A250 Hublift Rechts (EK1101)^A251 (EL1819)^Channel 4^.zyl_hublift_rechts_wt_einzug.fb.e_sensor1_ausgefahren} *)
	.zyl_hublift_rechts_wt_einzug.fb.e_sensor2_eingefahren AT %IX784.4 : BOOL;
	.zyl_hublift_rechts_wt_einzug.fb.e_sensor2_ausgefahren AT %IX784.5 : BOOL;
	.zyl_hublift_rechts_wt_einzug.fb.e_sensor3_eingefahren AT %IX784.6 : BOOL;
	.zyl_hublift_rechts_wt_einzug.fb.e_sensor3_ausgefahren AT %IX784.7 : BOOL;
	.zyl_hublift_rechts_wt_einzug.fb.e_sensor_mittegefahren AT %IX785.0 : BOOL;
	.zyl_hublift_rechts_wt_einzug.fb.e_taste_einfahren AT %IX785.1 : BOOL;
	.zyl_hublift_rechts_wt_einzug.fb.e_taste_ausfahren AT %IX785.2 : BOOL;
	.zyl_hublift_rechts_wt_einzug.fb.a_ventil_einfahren AT %QX743.5 : BOOL;	(*  ~ {LinkedWith:TIID^Gerät 1 (EtherCAT)^A250 Hublift Rechts (EK1101)^A253 (EL2809)^Channel 3^.zyl_hublift_rechts_wt_einzug.fb.a_ventil_einfahren} *)
	.zyl_hublift_rechts_wt_einzug.fb.a_ventil_ausfahren AT %QX743.6 : BOOL;	(*  ~ {LinkedWith:TIID^Gerät 1 (EtherCAT)^A250 Hublift Rechts (EK1101)^A253 (EL2809)^Channel 4^.zyl_hublift_rechts_wt_einzug.fb.a_ventil_ausfahren} *)
	.zyl_hublift_rechts_wt_klinke.fb.e_sensor1_eingefahren AT %IX785.3 : BOOL;	(*  ~ {LinkedWith:TIID^Gerät 1 (EtherCAT)^A250 Hublift Rechts (EK1101)^A251 (EL1819)^Channel 5^.zyl_hublift_rechts_wt_klinke.fb.e_sensor1_eingefahren} *)
	.zyl_hublift_rechts_wt_klinke.fb.e_sensor1_ausgefahren AT %IX785.4 : BOOL;	(*  ~ {LinkedWith:TIID^Gerät 1 (EtherCAT)^A250 Hublift Rechts (EK1101)^A251 (EL1819)^Channel 6^.zyl_hublift_rechts_wt_klinke.fb.e_sensor1_ausgefahren} *)
	.zyl_hublift_rechts_wt_klinke.fb.e_sensor2_eingefahren AT %IX785.5 : BOOL;
	.zyl_hublift_rechts_wt_klinke.fb.e_sensor2_ausgefahren AT %IX785.6 : BOOL;
	.zyl_hublift_rechts_wt_klinke.fb.e_sensor3_eingefahren AT %IX785.7 : BOOL;
	.zyl_hublift_rechts_wt_klinke.fb.e_sensor3_ausgefahren AT %IX786.0 : BOOL;
	.zyl_hublift_rechts_wt_klinke.fb.e_sensor_mittegefahren AT %IX786.1 : BOOL;
	.zyl_hublift_rechts_wt_klinke.fb.e_taste_einfahren AT %IX786.2 : BOOL;
	.zyl_hublift_rechts_wt_klinke.fb.e_taste_ausfahren AT %IX786.3 : BOOL;
	.zyl_hublift_rechts_wt_klinke.fb.a_ventil_einfahren AT %QX743.7 : BOOL;	(*  ~ {LinkedWith:TIID^Gerät 1 (EtherCAT)^A250 Hublift Rechts (EK1101)^A253 (EL2809)^Channel 5^.zyl_hublift_rechts_wt_klinke.fb.a_ventil_einfahren} *)
	.zyl_hublift_rechts_wt_klinke.fb.a_ventil_ausfahren AT %QX744.0 : BOOL;	(*  ~ {LinkedWith:TIID^Gerät 1 (EtherCAT)^A250 Hublift Rechts (EK1101)^A253 (EL2809)^Channel 6^.zyl_hublift_rechts_wt_klinke.fb.a_ventil_ausfahren} *)
	.zyl_hublift_links_lift.fb.e_sensor1_eingefahren AT %IX786.4 : BOOL;	(*  ~ {LinkedWith:TIID^Gerät 1 (EtherCAT)^A200 Hublift Links (EK1101)^A201 (EL1819)^Channel 1^.zyl_hublift_links_lift.fb.e_sensor1_eingefahren} *)
	.zyl_hublift_links_lift.fb.e_sensor1_ausgefahren AT %IX786.5 : BOOL;	(*  ~ {LinkedWith:TIID^Gerät 1 (EtherCAT)^A200 Hublift Links (EK1101)^A201 (EL1819)^Channel 2^.zyl_hublift_links_lift.fb.e_sensor1_ausgefahren} *)
	.zyl_hublift_links_lift.fb.e_sensor2_eingefahren AT %IX786.6 : BOOL;
	.zyl_hublift_links_lift.fb.e_sensor2_ausgefahren AT %IX786.7 : BOOL;
	.zyl_hublift_links_lift.fb.e_sensor3_eingefahren AT %IX787.0 : BOOL;
	.zyl_hublift_links_lift.fb.e_sensor3_ausgefahren AT %IX787.1 : BOOL;
	.zyl_hublift_links_lift.fb.e_sensor_mittegefahren AT %IX787.2 : BOOL;
	.zyl_hublift_links_lift.fb.e_taste_einfahren AT %IX787.3 : BOOL;
	.zyl_hublift_links_lift.fb.e_taste_ausfahren AT %IX787.4 : BOOL;
	.zyl_hublift_links_lift.fb.a_ventil_einfahren AT %QX744.1 : BOOL;	(*  ~ {LinkedWith:TIID^Gerät 1 (EtherCAT)^A200 Hublift Links (EK1101)^A203 (EL2809)^Channel 1^.zyl_hublift_links_lift.fb.a_ventil_einfahren} *)
	.zyl_hublift_links_lift.fb.a_ventil_ausfahren AT %QX744.2 : BOOL;	(*  ~ {LinkedWith:TIID^Gerät 1 (EtherCAT)^A200 Hublift Links (EK1101)^A203 (EL2809)^Channel 2^.zyl_hublift_links_lift.fb.a_ventil_ausfahren} *)
	.zyl_hublift_links_wt_einzug.fb.e_sensor1_eingefahren AT %IX787.5 : BOOL;	(*  ~ {LinkedWith:TIID^Gerät 1 (EtherCAT)^A200 Hublift Links (EK1101)^A201 (EL1819)^Channel 3^.zyl_hublift_links_wt_einzug.fb.e_sensor1_eingefahren} *)
	.zyl_hublift_links_wt_einzug.fb.e_sensor1_ausgefahren AT %IX787.6 : BOOL;	(*  ~ {LinkedWith:TIID^Gerät 1 (EtherCAT)^A200 Hublift Links (EK1101)^A201 (EL1819)^Channel 4^.zyl_hublift_links_wt_einzug.fb.e_sensor1_ausgefahren} *)
	.zyl_hublift_links_wt_einzug.fb.e_sensor2_eingefahren AT %IX787.7 : BOOL;
	.zyl_hublift_links_wt_einzug.fb.e_sensor2_ausgefahren AT %IX788.0 : BOOL;
	.zyl_hublift_links_wt_einzug.fb.e_sensor3_eingefahren AT %IX788.1 : BOOL;
	.zyl_hublift_links_wt_einzug.fb.e_sensor3_ausgefahren AT %IX788.2 : BOOL;
	.zyl_hublift_links_wt_einzug.fb.e_sensor_mittegefahren AT %IX788.3 : BOOL;
	.zyl_hublift_links_wt_einzug.fb.e_taste_einfahren AT %IX788.4 : BOOL;
	.zyl_hublift_links_wt_einzug.fb.e_taste_ausfahren AT %IX788.5 : BOOL;
	.zyl_hublift_links_wt_einzug.fb.a_ventil_einfahren AT %QX744.3 : BOOL;	(*  ~ {LinkedWith:TIID^Gerät 1 (EtherCAT)^A200 Hublift Links (EK1101)^A203 (EL2809)^Channel 3^.zyl_hublift_links_wt_einzug.fb.a_ventil_einfahren} *)
	.zyl_hublift_links_wt_einzug.fb.a_ventil_ausfahren AT %QX744.4 : BOOL;	(*  ~ {LinkedWith:TIID^Gerät 1 (EtherCAT)^A200 Hublift Links (EK1101)^A203 (EL2809)^Channel 4^.zyl_hublift_links_wt_einzug.fb.a_ventil_ausfahren} *)
	.zyl_hublift_links_wt_klinke.fb.e_sensor1_eingefahren AT %IX788.6 : BOOL;	(*  ~ {LinkedWith:TIID^Gerät 1 (EtherCAT)^A200 Hublift Links (EK1101)^A201 (EL1819)^Channel 5^.zyl_hublift_links_wt_klinke.fb.e_sensor1_eingefahren} *)
	.zyl_hublift_links_wt_klinke.fb.e_sensor1_ausgefahren AT %IX788.7 : BOOL;	(*  ~ {LinkedWith:TIID^Gerät 1 (EtherCAT)^A200 Hublift Links (EK1101)^A201 (EL1819)^Channel 6^.zyl_hublift_links_wt_klinke.fb.e_sensor1_ausgefahren} *)
	.zyl_hublift_links_wt_klinke.fb.e_sensor2_eingefahren AT %IX789.0 : BOOL;
	.zyl_hublift_links_wt_klinke.fb.e_sensor2_ausgefahren AT %IX789.1 : BOOL;
	.zyl_hublift_links_wt_klinke.fb.e_sensor3_eingefahren AT %IX789.2 : BOOL;
	.zyl_hublift_links_wt_klinke.fb.e_sensor3_ausgefahren AT %IX789.3 : BOOL;
	.zyl_hublift_links_wt_klinke.fb.e_sensor_mittegefahren AT %IX789.4 : BOOL;
	.zyl_hublift_links_wt_klinke.fb.e_taste_einfahren AT %IX789.5 : BOOL;
	.zyl_hublift_links_wt_klinke.fb.e_taste_ausfahren AT %IX789.6 : BOOL;
	.zyl_hublift_links_wt_klinke.fb.a_ventil_einfahren AT %QX744.5 : BOOL;	(*  ~ {LinkedWith:TIID^Gerät 1 (EtherCAT)^A200 Hublift Links (EK1101)^A203 (EL2809)^Channel 5^.zyl_hublift_links_wt_klinke.fb.a_ventil_einfahren} *)
	.zyl_hublift_links_wt_klinke.fb.a_ventil_ausfahren AT %QX744.6 : BOOL;	(*  ~ {LinkedWith:TIID^Gerät 1 (EtherCAT)^A200 Hublift Links (EK1101)^A203 (EL2809)^Channel 6^.zyl_hublift_links_wt_klinke.fb.a_ventil_ausfahren} *)
	.zyl_hublift_links_stopper.fb.e_sensor1_eingefahren AT %IX789.7 : BOOL;	(*  ~ {LinkedWith:TIID^Gerät 1 (EtherCAT)^A200 Hublift Links (EK1101)^A201 (EL1819)^Channel 7^.zyl_hublift_links_stopper.fb.e_sensor1_eingefahren} *)
	.zyl_hublift_links_stopper.fb.e_sensor1_ausgefahren AT %IX790.0 : BOOL;	(*  ~ {LinkedWith:TIID^Gerät 1 (EtherCAT)^A200 Hublift Links (EK1101)^A201 (EL1819)^Channel 8^.zyl_hublift_links_stopper.fb.e_sensor1_ausgefahren} *)
	.zyl_hublift_links_stopper.fb.e_sensor2_eingefahren AT %IX790.1 : BOOL;
	.zyl_hublift_links_stopper.fb.e_sensor2_ausgefahren AT %IX790.2 : BOOL;
	.zyl_hublift_links_stopper.fb.e_sensor3_eingefahren AT %IX790.3 : BOOL;
	.zyl_hublift_links_stopper.fb.e_sensor3_ausgefahren AT %IX790.4 : BOOL;
	.zyl_hublift_links_stopper.fb.e_sensor_mittegefahren AT %IX790.5 : BOOL;
	.zyl_hublift_links_stopper.fb.e_taste_einfahren AT %IX790.6 : BOOL;
	.zyl_hublift_links_stopper.fb.e_taste_ausfahren AT %IX790.7 : BOOL;
	.zyl_hublift_links_stopper.fb.a_ventil_einfahren AT %QX744.7 : BOOL;	(*  ~ {LinkedWith:TIID^Gerät 1 (EtherCAT)^A200 Hublift Links (EK1101)^A203 (EL2809)^Channel 7^.zyl_hublift_links_stopper.fb.a_ventil_einfahren} *)
	.zyl_hublift_links_stopper.fb.a_ventil_ausfahren AT %QX745.0 : BOOL;
	.zyl_hublift_links_eingriffschutz.fb.e_sensor1_eingefahren AT %IX1436.0 : BOOL;	(*  ~ {LinkedWith:TIID^Gerät 1 (EtherCAT)^A200 Hublift Links (EK1101)^A201 (EL1819)^Channel 11^.zyl_hublift_links_eingriffschutz.fb.e_sensor1_eingefahren} *)
	.zyl_hublift_links_eingriffschutz.fb.e_sensor1_ausgefahren AT %IX1436.1 : BOOL;	(*  ~ {LinkedWith:TIID^Gerät 1 (EtherCAT)^A200 Hublift Links (EK1101)^A201 (EL1819)^Channel 12^.zyl_hublift_links_eingriffschutz.fb.e_sensor1_ausgefahren} *)
	.zyl_hublift_links_eingriffschutz.fb.e_sensor2_eingefahren AT %IX1436.2 : BOOL;
	.zyl_hublift_links_eingriffschutz.fb.e_sensor2_ausgefahren AT %IX1436.3 : BOOL;
	.zyl_hublift_links_eingriffschutz.fb.e_sensor3_eingefahren AT %IX1436.4 : BOOL;
	.zyl_hublift_links_eingriffschutz.fb.e_sensor3_ausgefahren AT %IX1436.5 : BOOL;
	.zyl_hublift_links_eingriffschutz.fb.e_sensor_mittegefahren AT %IX1436.6 : BOOL;
	.zyl_hublift_links_eingriffschutz.fb.e_taste_einfahren AT %IX1436.7 : BOOL;
	.zyl_hublift_links_eingriffschutz.fb.e_taste_ausfahren AT %IX1437.0 : BOOL;
	.zyl_hublift_links_eingriffschutz.fb.a_ventil_einfahren AT %QX1305.0 : BOOL;	(*  ~ {LinkedWith:TIID^Gerät 1 (EtherCAT)^A200 Hublift Links (EK1101)^A203 (EL2809)^Channel 9^.zyl_hublift_links_eingriffschutz.fb.a_ventil_einfahren} *)
	.zyl_hublift_links_eingriffschutz.fb.a_ventil_ausfahren AT %QX1305.1 : BOOL;	(*  ~ {LinkedWith:TIID^Gerät 1 (EtherCAT)^A200 Hublift Links (EK1101)^A203 (EL2809)^Channel 10^.zyl_hublift_links_eingriffschutz.fb.a_ventil_ausfahren} *)
	.zyl_bandfaenger.fb.e_sensor1_eingefahren AT %IX791.0 : BOOL;
	.zyl_bandfaenger.fb.e_sensor1_ausgefahren AT %IX791.1 : BOOL;	(*  ~ {LinkedWith:TIID^Gerät 1 (EtherCAT)^A150 (EP2338-0001)^Channel 5^.zyl_bandfaenger.fb.e_sensor1_ausgefahren} *)
	.zyl_bandfaenger.fb.e_sensor2_eingefahren AT %IX791.2 : BOOL;
	.zyl_bandfaenger.fb.e_sensor2_ausgefahren AT %IX791.3 : BOOL;
	.zyl_bandfaenger.fb.e_sensor3_eingefahren AT %IX791.4 : BOOL;
	.zyl_bandfaenger.fb.e_sensor3_ausgefahren AT %IX791.5 : BOOL;
	.zyl_bandfaenger.fb.e_sensor_mittegefahren AT %IX791.6 : BOOL;
	.zyl_bandfaenger.fb.e_taste_einfahren AT %IX791.7 : BOOL;
	.zyl_bandfaenger.fb.e_taste_ausfahren AT %IX792.0 : BOOL;
	.zyl_bandfaenger.fb.a_ventil_einfahren AT %QX745.1 : BOOL;
	.zyl_bandfaenger.fb.a_ventil_ausfahren AT %QX745.2 : BOOL;
	.zyl_bandklemmen.fb.e_sensor1_eingefahren AT %IX792.1 : BOOL;
	.zyl_bandklemmen.fb.e_sensor1_ausgefahren AT %IX792.2 : BOOL;	(*  ~ {LinkedWith:TIID^Gerät 1 (EtherCAT)^A150 (EP2338-0001)^Channel 6^.zyl_bandklemmen.fb.e_sensor1_ausgefahren} *)
	.zyl_bandklemmen.fb.e_sensor2_eingefahren AT %IX792.3 : BOOL;
	.zyl_bandklemmen.fb.e_sensor2_ausgefahren AT %IX792.4 : BOOL;
	.zyl_bandklemmen.fb.e_sensor3_eingefahren AT %IX792.5 : BOOL;
	.zyl_bandklemmen.fb.e_sensor3_ausgefahren AT %IX792.6 : BOOL;
	.zyl_bandklemmen.fb.e_sensor_mittegefahren AT %IX792.7 : BOOL;
	.zyl_bandklemmen.fb.e_taste_einfahren AT %IX793.0 : BOOL;
	.zyl_bandklemmen.fb.e_taste_ausfahren AT %IX793.1 : BOOL;
	.zyl_bandklemmen.fb.a_ventil_einfahren AT %QX745.3 : BOOL;
	.zyl_bandklemmen.fb.a_ventil_ausfahren AT %QX745.4 : BOOL;
	.zyl_bawe_vorschub.fb.e_sensor1_eingefahren AT %IX793.2 : BOOL;	(*  ~ {LinkedWith:TIID^Gerät 1 (EtherCAT)^A160 (EP2338-0001)^Channel 5^.zyl_bawe_vorschub.fb.e_sensor1_eingefahren} *)
	.zyl_bawe_vorschub.fb.e_sensor1_ausgefahren AT %IX793.3 : BOOL;	(*  ~ {LinkedWith:TIID^Gerät 1 (EtherCAT)^A160 (EP2338-0001)^Channel 6^.zyl_bawe_vorschub.fb.e_sensor1_ausgefahren} *)
	.zyl_bawe_vorschub.fb.e_sensor2_eingefahren AT %IX793.4 : BOOL;
	.zyl_bawe_vorschub.fb.e_sensor2_ausgefahren AT %IX793.5 : BOOL;
	.zyl_bawe_vorschub.fb.e_sensor3_eingefahren AT %IX793.6 : BOOL;
	.zyl_bawe_vorschub.fb.e_sensor3_ausgefahren AT %IX793.7 : BOOL;
	.zyl_bawe_vorschub.fb.e_sensor_mittegefahren AT %IX794.0 : BOOL;
	.zyl_bawe_vorschub.fb.e_taste_einfahren AT %IX794.1 : BOOL;
	.zyl_bawe_vorschub.fb.e_taste_ausfahren AT %IX794.2 : BOOL;
	.zyl_bawe_vorschub.fb.a_ventil_einfahren AT %QX745.5 : BOOL;
	.zyl_bawe_vorschub.fb.a_ventil_ausfahren AT %QX745.6 : BOOL;
	.zyl_bawe_querschub.fb.e_sensor1_eingefahren AT %IX794.3 : BOOL;	(*  ~ {LinkedWith:TIID^Gerät 1 (EtherCAT)^A160 (EP2338-0001)^Channel 7^.zyl_bawe_querschub.fb.e_sensor1_eingefahren} *)
	.zyl_bawe_querschub.fb.e_sensor1_ausgefahren AT %IX794.4 : BOOL;	(*  ~ {LinkedWith:TIID^Gerät 1 (EtherCAT)^A160 (EP2338-0001)^Channel 8^.zyl_bawe_querschub.fb.e_sensor1_ausgefahren} *)
	.zyl_bawe_querschub.fb.e_sensor2_eingefahren AT %IX794.5 : BOOL;
	.zyl_bawe_querschub.fb.e_sensor2_ausgefahren AT %IX794.6 : BOOL;
	.zyl_bawe_querschub.fb.e_sensor3_eingefahren AT %IX794.7 : BOOL;
	.zyl_bawe_querschub.fb.e_sensor3_ausgefahren AT %IX795.0 : BOOL;
	.zyl_bawe_querschub.fb.e_sensor_mittegefahren AT %IX795.1 : BOOL;
	.zyl_bawe_querschub.fb.e_taste_einfahren AT %IX795.2 : BOOL;
	.zyl_bawe_querschub.fb.e_taste_ausfahren AT %IX795.3 : BOOL;
	.zyl_bawe_querschub.fb.a_ventil_einfahren AT %QX745.7 : BOOL;	(*  ~ {LinkedWith:TIID^Gerät 1 (EtherCAT)^A50 (CPX-FB38 64Byte)^Outputs^QB4^.zyl_bawe_querschub.fb.a_ventil_einfahren} *)
	.zyl_bawe_querschub.fb.a_ventil_ausfahren AT %QX746.0 : BOOL;	(*  ~ {LinkedWith:TIID^Gerät 1 (EtherCAT)^A50 (CPX-FB38 64Byte)^Outputs^QB4^.zyl_bawe_querschub.fb.a_ventil_ausfahren} *)
	.zyl_bawe_faenger_li.fb.e_sensor1_eingefahren AT %IX795.4 : BOOL;
	.zyl_bawe_faenger_li.fb.e_sensor1_ausgefahren AT %IX795.5 : BOOL;
	.zyl_bawe_faenger_li.fb.e_sensor2_eingefahren AT %IX795.6 : BOOL;
	.zyl_bawe_faenger_li.fb.e_sensor2_ausgefahren AT %IX795.7 : BOOL;
	.zyl_bawe_faenger_li.fb.e_sensor3_eingefahren AT %IX796.0 : BOOL;
	.zyl_bawe_faenger_li.fb.e_sensor3_ausgefahren AT %IX796.1 : BOOL;
	.zyl_bawe_faenger_li.fb.e_sensor_mittegefahren AT %IX796.2 : BOOL;
	.zyl_bawe_faenger_li.fb.e_taste_einfahren AT %IX796.3 : BOOL;
	.zyl_bawe_faenger_li.fb.e_taste_ausfahren AT %IX796.4 : BOOL;
	.zyl_bawe_faenger_li.fb.a_ventil_einfahren AT %QX746.1 : BOOL;	(*  ~ {LinkedWith:TIID^Gerät 1 (EtherCAT)^A50 (CPX-FB38 64Byte)^Outputs^QB3^.zyl_bawe_faenger_li.fb.a_ventil_einfahren} *)
	.zyl_bawe_faenger_li.fb.a_ventil_ausfahren AT %QX746.2 : BOOL;	(*  ~ {LinkedWith:TIID^Gerät 1 (EtherCAT)^A50 (CPX-FB38 64Byte)^Outputs^QB3^.zyl_bawe_faenger_li.fb.a_ventil_ausfahren} *)
	.zyl_bawe_faenger_re.fb.e_sensor1_eingefahren AT %IX796.5 : BOOL;
	.zyl_bawe_faenger_re.fb.e_sensor1_ausgefahren AT %IX796.6 : BOOL;
	.zyl_bawe_faenger_re.fb.e_sensor2_eingefahren AT %IX796.7 : BOOL;
	.zyl_bawe_faenger_re.fb.e_sensor2_ausgefahren AT %IX797.0 : BOOL;
	.zyl_bawe_faenger_re.fb.e_sensor3_eingefahren AT %IX797.1 : BOOL;
	.zyl_bawe_faenger_re.fb.e_sensor3_ausgefahren AT %IX797.2 : BOOL;
	.zyl_bawe_faenger_re.fb.e_sensor_mittegefahren AT %IX797.3 : BOOL;
	.zyl_bawe_faenger_re.fb.e_taste_einfahren AT %IX797.4 : BOOL;
	.zyl_bawe_faenger_re.fb.e_taste_ausfahren AT %IX797.5 : BOOL;
	.zyl_bawe_faenger_re.fb.a_ventil_einfahren AT %QX746.3 : BOOL;	(*  ~ {LinkedWith:TIID^Gerät 1 (EtherCAT)^A50 (CPX-FB38 64Byte)^Outputs^QB3^.zyl_bawe_faenger_re.fb.a_ventil_einfahren} *)
	.zyl_bawe_faenger_re.fb.a_ventil_ausfahren AT %QX746.4 : BOOL;	(*  ~ {LinkedWith:TIID^Gerät 1 (EtherCAT)^A50 (CPX-FB38 64Byte)^Outputs^QB3^.zyl_bawe_faenger_re.fb.a_ventil_ausfahren} *)
	.zyl_bawe_halter_li.fb.e_sensor1_eingefahren AT %IX797.6 : BOOL;
	.zyl_bawe_halter_li.fb.e_sensor1_ausgefahren AT %IX797.7 : BOOL;
	.zyl_bawe_halter_li.fb.e_sensor2_eingefahren AT %IX798.0 : BOOL;
	.zyl_bawe_halter_li.fb.e_sensor2_ausgefahren AT %IX798.1 : BOOL;
	.zyl_bawe_halter_li.fb.e_sensor3_eingefahren AT %IX798.2 : BOOL;
	.zyl_bawe_halter_li.fb.e_sensor3_ausgefahren AT %IX798.3 : BOOL;
	.zyl_bawe_halter_li.fb.e_sensor_mittegefahren AT %IX798.4 : BOOL;
	.zyl_bawe_halter_li.fb.e_taste_einfahren AT %IX798.5 : BOOL;
	.zyl_bawe_halter_li.fb.e_taste_ausfahren AT %IX798.6 : BOOL;
	.zyl_bawe_halter_li.fb.a_ventil_einfahren AT %QX746.5 : BOOL;	(*  ~ {LinkedWith:TIID^Gerät 1 (EtherCAT)^A50 (CPX-FB38 64Byte)^Outputs^QB3^.zyl_bawe_halter_li.fb.a_ventil_einfahren} *)
	.zyl_bawe_halter_li.fb.a_ventil_ausfahren AT %QX746.6 : BOOL;	(*  ~ {LinkedWith:TIID^Gerät 1 (EtherCAT)^A50 (CPX-FB38 64Byte)^Outputs^QB3^.zyl_bawe_halter_li.fb.a_ventil_ausfahren} *)
	.zyl_bawe_halter_re.fb.e_sensor1_eingefahren AT %IX798.7 : BOOL;
	.zyl_bawe_halter_re.fb.e_sensor1_ausgefahren AT %IX799.0 : BOOL;
	.zyl_bawe_halter_re.fb.e_sensor2_eingefahren AT %IX799.1 : BOOL;
	.zyl_bawe_halter_re.fb.e_sensor2_ausgefahren AT %IX799.2 : BOOL;
	.zyl_bawe_halter_re.fb.e_sensor3_eingefahren AT %IX799.3 : BOOL;
	.zyl_bawe_halter_re.fb.e_sensor3_ausgefahren AT %IX799.4 : BOOL;
	.zyl_bawe_halter_re.fb.e_sensor_mittegefahren AT %IX799.5 : BOOL;
	.zyl_bawe_halter_re.fb.e_taste_einfahren AT %IX799.6 : BOOL;
	.zyl_bawe_halter_re.fb.e_taste_ausfahren AT %IX799.7 : BOOL;
	.zyl_bawe_halter_re.fb.a_ventil_einfahren AT %QX746.7 : BOOL;	(*  ~ {LinkedWith:TIID^Gerät 1 (EtherCAT)^A50 (CPX-FB38 64Byte)^Outputs^QB3^.zyl_bawe_halter_re.fb.a_ventil_einfahren} *)
	.zyl_bawe_halter_re.fb.a_ventil_ausfahren AT %QX747.0 : BOOL;	(*  ~ {LinkedWith:TIID^Gerät 1 (EtherCAT)^A50 (CPX-FB38 64Byte)^Outputs^QB3^.zyl_bawe_halter_re.fb.a_ventil_ausfahren} *)
	.zyl_haspel_verschieben.fb.e_sensor1_eingefahren AT %IX800.0 : BOOL;	(*  ~ {LinkedWith:TIID^Gerät 1 (EtherCAT)^A38 Transportsystem (EP2338-0001)^Channel 2^.zyl_haspel_verschieben.fb.e_sensor1_eingefahren} *)
	.zyl_haspel_verschieben.fb.e_sensor1_ausgefahren AT %IX800.1 : BOOL;	(*  ~ {LinkedWith:TIID^Gerät 1 (EtherCAT)^A38 Transportsystem (EP2338-0001)^Channel 1^.zyl_haspel_verschieben.fb.e_sensor1_ausgefahren} *)
	.zyl_haspel_verschieben.fb.e_sensor2_eingefahren AT %IX800.2 : BOOL;
	.zyl_haspel_verschieben.fb.e_sensor2_ausgefahren AT %IX800.3 : BOOL;
	.zyl_haspel_verschieben.fb.e_sensor3_eingefahren AT %IX800.4 : BOOL;
	.zyl_haspel_verschieben.fb.e_sensor3_ausgefahren AT %IX800.5 : BOOL;
	.zyl_haspel_verschieben.fb.e_sensor_mittegefahren AT %IX800.6 : BOOL;
	.zyl_haspel_verschieben.fb.e_taste_einfahren AT %IX800.7 : BOOL;
	.zyl_haspel_verschieben.fb.e_taste_ausfahren AT %IX801.0 : BOOL;
	.zyl_haspel_verschieben.fb.a_ventil_einfahren AT %QX747.1 : BOOL;	(*  ~ {LinkedWith:TIID^Gerät 1 (EtherCAT)^Schaltschrank (EK1100)^A46 (EL2809)^Channel 11^.zyl_haspel_verschieben.fb.a_ventil_einfahren} *)
	.zyl_haspel_verschieben.fb.a_ventil_ausfahren AT %QX747.2 : BOOL;	(*  ~ {LinkedWith:TIID^Gerät 1 (EtherCAT)^Schaltschrank (EK1100)^A46 (EL2809)^Channel 12^.zyl_haspel_verschieben.fb.a_ventil_ausfahren} *)
	.zyl_bandeinzuege_verschieben.fb.e_sensor1_eingefahren AT %IX801.1 : BOOL;	(*  ~ {LinkedWith:TIID^Gerät 1 (EtherCAT)^A38 Transportsystem (EP2338-0001)^Channel 3^.zyl_bandeinzuege_verschieben.fb.e_sensor1_eingefahren} *)
	.zyl_bandeinzuege_verschieben.fb.e_sensor1_ausgefahren AT %IX801.2 : BOOL;	(*  ~ {LinkedWith:TIID^Gerät 1 (EtherCAT)^A38 Transportsystem (EP2338-0001)^Channel 4^.zyl_bandeinzuege_verschieben.fb.e_sensor1_ausgefahren} *)
	.zyl_bandeinzuege_verschieben.fb.e_sensor2_eingefahren AT %IX801.3 : BOOL;
	.zyl_bandeinzuege_verschieben.fb.e_sensor2_ausgefahren AT %IX801.4 : BOOL;
	.zyl_bandeinzuege_verschieben.fb.e_sensor3_eingefahren AT %IX801.5 : BOOL;
	.zyl_bandeinzuege_verschieben.fb.e_sensor3_ausgefahren AT %IX801.6 : BOOL;
	.zyl_bandeinzuege_verschieben.fb.e_sensor_mittegefahren AT %IX801.7 : BOOL;
	.zyl_bandeinzuege_verschieben.fb.e_taste_einfahren AT %IX802.0 : BOOL;
	.zyl_bandeinzuege_verschieben.fb.e_taste_ausfahren AT %IX802.1 : BOOL;
	.zyl_bandeinzuege_verschieben.fb.a_ventil_einfahren AT %QX747.3 : BOOL;	(*  ~ {LinkedWith:TIID^Gerät 1 (EtherCAT)^A50 (CPX-FB38 64Byte)^Outputs^QB1^.zyl_bandeinzuege_verschieben.fb.a_ventil_einfahren} *)
	.zyl_bandeinzuege_verschieben.fb.a_ventil_ausfahren AT %QX747.4 : BOOL;	(*  ~ {LinkedWith:TIID^Gerät 1 (EtherCAT)^A50 (CPX-FB38 64Byte)^Outputs^QB1^.zyl_bandeinzuege_verschieben.fb.a_ventil_ausfahren} *)
	.zyl_oelen_unten.fb.e_sensor1_eingefahren AT %IX1437.1 : BOOL;	(*  ~ {LinkedWith:TIID^Gerät 1 (EtherCAT)^A170 (EP2338-0001)^Channel 3^.zyl_oelen_unten.fb.e_sensor1_eingefahren} *)
	.zyl_oelen_unten.fb.e_sensor1_ausgefahren AT %IX1437.2 : BOOL;	(*  ~ {LinkedWith:TIID^Gerät 1 (EtherCAT)^A170 (EP2338-0001)^Channel 4^.zyl_oelen_unten.fb.e_sensor1_ausgefahren} *)
	.zyl_oelen_unten.fb.e_sensor2_eingefahren AT %IX1437.3 : BOOL;
	.zyl_oelen_unten.fb.e_sensor2_ausgefahren AT %IX1437.4 : BOOL;
	.zyl_oelen_unten.fb.e_sensor3_eingefahren AT %IX1437.5 : BOOL;
	.zyl_oelen_unten.fb.e_sensor3_ausgefahren AT %IX1437.6 : BOOL;
	.zyl_oelen_unten.fb.e_sensor_mittegefahren AT %IX1437.7 : BOOL;
	.zyl_oelen_unten.fb.e_taste_einfahren AT %IX1438.0 : BOOL;
	.zyl_oelen_unten.fb.e_taste_ausfahren AT %IX1438.1 : BOOL;
	.zyl_oelen_unten.fb.a_ventil_einfahren AT %QX1305.2 : BOOL;
	.zyl_oelen_unten.fb.a_ventil_ausfahren AT %QX1305.3 : BOOL;	(*  ~ {LinkedWith:TIID^Gerät 1 (EtherCAT)^A170 (EP2338-0001)^Channel 14^.zyl_oelen_unten.fb.a_ventil_ausfahren} *)
	.zyl_oelen_oben.fb.e_sensor1_eingefahren AT %IX1438.2 : BOOL;	(*  ~ {LinkedWith:TIID^Gerät 1 (EtherCAT)^A170 (EP2338-0001)^Channel 1^.zyl_oelen_oben.fb.e_sensor1_eingefahren} *)
	.zyl_oelen_oben.fb.e_sensor1_ausgefahren AT %IX1438.3 : BOOL;	(*  ~ {LinkedWith:TIID^Gerät 1 (EtherCAT)^A170 (EP2338-0001)^Channel 2^.zyl_oelen_oben.fb.e_sensor1_ausgefahren} *)
	.zyl_oelen_oben.fb.e_sensor2_eingefahren AT %IX1438.4 : BOOL;
	.zyl_oelen_oben.fb.e_sensor2_ausgefahren AT %IX1438.5 : BOOL;
	.zyl_oelen_oben.fb.e_sensor3_eingefahren AT %IX1438.6 : BOOL;
	.zyl_oelen_oben.fb.e_sensor3_ausgefahren AT %IX1438.7 : BOOL;
	.zyl_oelen_oben.fb.e_sensor_mittegefahren AT %IX1439.0 : BOOL;
	.zyl_oelen_oben.fb.e_taste_einfahren AT %IX1439.1 : BOOL;
	.zyl_oelen_oben.fb.e_taste_ausfahren AT %IX1439.2 : BOOL;
	.zyl_oelen_oben.fb.a_ventil_einfahren AT %QX1305.4 : BOOL;
	.zyl_oelen_oben.fb.a_ventil_ausfahren AT %QX1305.5 : BOOL;	(*  ~ {LinkedWith:TIID^Gerät 1 (EtherCAT)^A170 (EP2338-0001)^Channel 13^.zyl_oelen_oben.fb.a_ventil_ausfahren} *)
	.zyl_Indexier_Bestueckpos.fb.e_sensor1_eingefahren AT %IX1576.0 : BOOL;
	.zyl_Indexier_Bestueckpos.fb.e_sensor1_ausgefahren AT %IX1576.1 : BOOL;
	.zyl_Indexier_Bestueckpos.fb.e_sensor2_eingefahren AT %IX1576.2 : BOOL;
	.zyl_Indexier_Bestueckpos.fb.e_sensor2_ausgefahren AT %IX1576.3 : BOOL;
	.zyl_Indexier_Bestueckpos.fb.e_sensor3_eingefahren AT %IX1576.4 : BOOL;
	.zyl_Indexier_Bestueckpos.fb.e_sensor3_ausgefahren AT %IX1576.5 : BOOL;
	.zyl_Indexier_Bestueckpos.fb.e_sensor_mittegefahren AT %IX1576.6 : BOOL;
	.zyl_Indexier_Bestueckpos.fb.e_taste_einfahren AT %IX1576.7 : BOOL;
	.zyl_Indexier_Bestueckpos.fb.e_taste_ausfahren AT %IX1577.0 : BOOL;
	.zyl_Indexier_Bestueckpos.fb.a_ventil_einfahren AT %QX1437.0 : BOOL;
	.zyl_Indexier_Bestueckpos.fb.a_ventil_ausfahren AT %QX1437.1 : BOOL;
	.zyl_Indexier_Einlauf.fb.e_sensor1_eingefahren AT %IX1577.1 : BOOL;
	.zyl_Indexier_Einlauf.fb.e_sensor1_ausgefahren AT %IX1577.2 : BOOL;
	.zyl_Indexier_Einlauf.fb.e_sensor2_eingefahren AT %IX1577.3 : BOOL;
	.zyl_Indexier_Einlauf.fb.e_sensor2_ausgefahren AT %IX1577.4 : BOOL;
	.zyl_Indexier_Einlauf.fb.e_sensor3_eingefahren AT %IX1577.5 : BOOL;
	.zyl_Indexier_Einlauf.fb.e_sensor3_ausgefahren AT %IX1577.6 : BOOL;
	.zyl_Indexier_Einlauf.fb.e_sensor_mittegefahren AT %IX1577.7 : BOOL;
	.zyl_Indexier_Einlauf.fb.e_taste_einfahren AT %IX1578.0 : BOOL;
	.zyl_Indexier_Einlauf.fb.e_taste_ausfahren AT %IX1578.1 : BOOL;
	.zyl_Indexier_Einlauf.fb.a_ventil_einfahren AT %QX1437.2 : BOOL;
	.zyl_Indexier_Einlauf.fb.a_ventil_ausfahren AT %QX1437.3 : BOOL;
	.zyl_wt_stopper_einlauf.fb.e_sensor1_eingefahren AT %IX807.7 : BOOL;
	.zyl_wt_stopper_einlauf.fb.e_sensor1_ausgefahren AT %IX808.0 : BOOL;
	.zyl_wt_stopper_einlauf.fb.e_sensor2_eingefahren AT %IX808.1 : BOOL;
	.zyl_wt_stopper_einlauf.fb.e_sensor2_ausgefahren AT %IX808.2 : BOOL;
	.zyl_wt_stopper_einlauf.fb.e_sensor3_eingefahren AT %IX808.3 : BOOL;
	.zyl_wt_stopper_einlauf.fb.e_sensor3_ausgefahren AT %IX808.4 : BOOL;
	.zyl_wt_stopper_einlauf.fb.e_sensor_mittegefahren AT %IX808.5 : BOOL;
	.zyl_wt_stopper_einlauf.fb.e_taste_einfahren AT %IX808.6 : BOOL;
	.zyl_wt_stopper_einlauf.fb.e_taste_ausfahren AT %IX808.7 : BOOL;
	.zyl_wt_stopper_einlauf.fb.a_ventil_einfahren AT %QX748.7 : BOOL;	(*  ~ {LinkedWith:TIID^Gerät 1 (EtherCAT)^A50 (CPX-FB38 64Byte)^Outputs^QB0^.zyl_wt_stopper_einlauf.fb.a_ventil_einfahren} *)
	.zyl_wt_stopper_einlauf.fb.a_ventil_ausfahren AT %QX749.0 : BOOL;
	.zyl_bandfaenger_li.fb.e_sensor1_eingefahren AT %IX809.0 : BOOL;
	.zyl_bandfaenger_li.fb.e_sensor1_ausgefahren AT %IX809.1 : BOOL;
	.zyl_bandfaenger_li.fb.e_sensor2_eingefahren AT %IX809.2 : BOOL;
	.zyl_bandfaenger_li.fb.e_sensor2_ausgefahren AT %IX809.3 : BOOL;
	.zyl_bandfaenger_li.fb.e_sensor3_eingefahren AT %IX809.4 : BOOL;
	.zyl_bandfaenger_li.fb.e_sensor3_ausgefahren AT %IX809.5 : BOOL;
	.zyl_bandfaenger_li.fb.e_sensor_mittegefahren AT %IX809.6 : BOOL;
	.zyl_bandfaenger_li.fb.e_taste_einfahren AT %IX809.7 : BOOL;
	.zyl_bandfaenger_li.fb.e_taste_ausfahren AT %IX810.0 : BOOL;
	.zyl_bandfaenger_li.fb.a_ventil_einfahren AT %QX749.1 : BOOL;
	.zyl_bandfaenger_li.fb.a_ventil_ausfahren AT %QX749.2 : BOOL;
	.zyl_bandfaenger_re.fb.e_sensor1_eingefahren AT %IX810.1 : BOOL;
	.zyl_bandfaenger_re.fb.e_sensor1_ausgefahren AT %IX810.2 : BOOL;
	.zyl_bandfaenger_re.fb.e_sensor2_eingefahren AT %IX810.3 : BOOL;
	.zyl_bandfaenger_re.fb.e_sensor2_ausgefahren AT %IX810.4 : BOOL;
	.zyl_bandfaenger_re.fb.e_sensor3_eingefahren AT %IX810.5 : BOOL;
	.zyl_bandfaenger_re.fb.e_sensor3_ausgefahren AT %IX810.6 : BOOL;
	.zyl_bandfaenger_re.fb.e_sensor_mittegefahren AT %IX810.7 : BOOL;
	.zyl_bandfaenger_re.fb.e_taste_einfahren AT %IX811.0 : BOOL;
	.zyl_bandfaenger_re.fb.e_taste_ausfahren AT %IX811.1 : BOOL;
	.zyl_bandfaenger_re.fb.a_ventil_einfahren AT %QX749.3 : BOOL;
	.zyl_bandfaenger_re.fb.a_ventil_ausfahren AT %QX749.4 : BOOL;
	.zyl_bandklemmen_li.fb.e_sensor1_eingefahren AT %IX811.2 : BOOL;
	.zyl_bandklemmen_li.fb.e_sensor1_ausgefahren AT %IX811.3 : BOOL;
	.zyl_bandklemmen_li.fb.e_sensor2_eingefahren AT %IX811.4 : BOOL;
	.zyl_bandklemmen_li.fb.e_sensor2_ausgefahren AT %IX811.5 : BOOL;
	.zyl_bandklemmen_li.fb.e_sensor3_eingefahren AT %IX811.6 : BOOL;
	.zyl_bandklemmen_li.fb.e_sensor3_ausgefahren AT %IX811.7 : BOOL;
	.zyl_bandklemmen_li.fb.e_sensor_mittegefahren AT %IX812.0 : BOOL;
	.zyl_bandklemmen_li.fb.e_taste_einfahren AT %IX812.1 : BOOL;
	.zyl_bandklemmen_li.fb.e_taste_ausfahren AT %IX812.2 : BOOL;
	.zyl_bandklemmen_li.fb.a_ventil_einfahren AT %QX749.5 : BOOL;
	.zyl_bandklemmen_li.fb.a_ventil_ausfahren AT %QX749.6 : BOOL;
	.zyl_bandklemmen_re.fb.e_sensor1_eingefahren AT %IX812.3 : BOOL;
	.zyl_bandklemmen_re.fb.e_sensor1_ausgefahren AT %IX812.4 : BOOL;
	.zyl_bandklemmen_re.fb.e_sensor2_eingefahren AT %IX812.5 : BOOL;
	.zyl_bandklemmen_re.fb.e_sensor2_ausgefahren AT %IX812.6 : BOOL;
	.zyl_bandklemmen_re.fb.e_sensor3_eingefahren AT %IX812.7 : BOOL;
	.zyl_bandklemmen_re.fb.e_sensor3_ausgefahren AT %IX813.0 : BOOL;
	.zyl_bandklemmen_re.fb.e_sensor_mittegefahren AT %IX813.1 : BOOL;
	.zyl_bandklemmen_re.fb.e_taste_einfahren AT %IX813.2 : BOOL;
	.zyl_bandklemmen_re.fb.e_taste_ausfahren AT %IX813.3 : BOOL;
	.zyl_bandklemmen_re.fb.a_ventil_einfahren AT %QX749.7 : BOOL;
	.zyl_bandklemmen_re.fb.a_ventil_ausfahren AT %QX750.0 : BOOL;
	.zyl_rafo_faenger.fb.e_sensor1_eingefahren AT %IX813.4 : BOOL;
	.zyl_rafo_faenger.fb.e_sensor1_ausgefahren AT %IX813.5 : BOOL;	(*  ~ {LinkedWith:TIID^Gerät 1 (EtherCAT)^A150 (EP2338-0001)^Channel 5^.zyl_bandfaenger.fb.e_sensor1_ausgefahren} *)
	.zyl_rafo_faenger.fb.e_sensor2_eingefahren AT %IX813.6 : BOOL;
	.zyl_rafo_faenger.fb.e_sensor2_ausgefahren AT %IX813.7 : BOOL;
	.zyl_rafo_faenger.fb.e_sensor3_eingefahren AT %IX814.0 : BOOL;
	.zyl_rafo_faenger.fb.e_sensor3_ausgefahren AT %IX814.1 : BOOL;
	.zyl_rafo_faenger.fb.e_sensor_mittegefahren AT %IX814.2 : BOOL;
	.zyl_rafo_faenger.fb.e_taste_einfahren AT %IX814.3 : BOOL;
	.zyl_rafo_faenger.fb.e_taste_ausfahren AT %IX814.4 : BOOL;
	.zyl_rafo_faenger.fb.a_ventil_einfahren AT %QX750.1 : BOOL;
	.zyl_rafo_faenger.fb.a_ventil_ausfahren AT %QX750.2 : BOOL;
	.zyl_rafo_klemmen.fb.e_sensor1_eingefahren AT %IX814.5 : BOOL;
	.zyl_rafo_klemmen.fb.e_sensor1_ausgefahren AT %IX814.6 : BOOL;	(*  ~ {LinkedWith:TIID^Gerät 1 (EtherCAT)^A150 (EP2338-0001)^Channel 6^.zyl_bandklemmen.fb.e_sensor1_ausgefahren} *)
	.zyl_rafo_klemmen.fb.e_sensor2_eingefahren AT %IX814.7 : BOOL;
	.zyl_rafo_klemmen.fb.e_sensor2_ausgefahren AT %IX815.0 : BOOL;
	.zyl_rafo_klemmen.fb.e_sensor3_eingefahren AT %IX815.1 : BOOL;
	.zyl_rafo_klemmen.fb.e_sensor3_ausgefahren AT %IX815.2 : BOOL;
	.zyl_rafo_klemmen.fb.e_sensor_mittegefahren AT %IX815.3 : BOOL;
	.zyl_rafo_klemmen.fb.e_taste_einfahren AT %IX815.4 : BOOL;
	.zyl_rafo_klemmen.fb.e_taste_ausfahren AT %IX815.5 : BOOL;
	.zyl_rafo_klemmen.fb.a_ventil_einfahren AT %QX750.3 : BOOL;
	.zyl_rafo_klemmen.fb.a_ventil_ausfahren AT %QX750.4 : BOOL;
	.zyl_rafo_vorschub.fb.e_sensor1_eingefahren AT %IX815.6 : BOOL;	(*  ~ {LinkedWith:TIID^Gerät 1 (EtherCAT)^A160 (EP2338-0001)^Channel 5^.zyl_bawe_vorschub.fb.e_sensor1_eingefahren} *)
	.zyl_rafo_vorschub.fb.e_sensor1_ausgefahren AT %IX815.7 : BOOL;	(*  ~ {LinkedWith:TIID^Gerät 1 (EtherCAT)^A160 (EP2338-0001)^Channel 6^.zyl_bawe_vorschub.fb.e_sensor1_ausgefahren} *)
	.zyl_rafo_vorschub.fb.e_sensor2_eingefahren AT %IX816.0 : BOOL;
	.zyl_rafo_vorschub.fb.e_sensor2_ausgefahren AT %IX816.1 : BOOL;
	.zyl_rafo_vorschub.fb.e_sensor3_eingefahren AT %IX816.2 : BOOL;
	.zyl_rafo_vorschub.fb.e_sensor3_ausgefahren AT %IX816.3 : BOOL;
	.zyl_rafo_vorschub.fb.e_sensor_mittegefahren AT %IX816.4 : BOOL;
	.zyl_rafo_vorschub.fb.e_taste_einfahren AT %IX816.5 : BOOL;
	.zyl_rafo_vorschub.fb.e_taste_ausfahren AT %IX816.6 : BOOL;
	.zyl_rafo_vorschub.fb.a_ventil_einfahren AT %QX750.5 : BOOL;
	.zyl_rafo_vorschub.fb.a_ventil_ausfahren AT %QX750.6 : BOOL;
	.zyl_rafo_kamm.fb.e_sensor1_eingefahren AT %IX816.7 : BOOL;	(*  ~ {LinkedWith:TIID^Gerät 1 (EtherCAT)^A160 (EP2338-0001)^Channel 1^.zyl_rafo_kamm.fb.e_sensor1_eingefahren} *)
	.zyl_rafo_kamm.fb.e_sensor1_ausgefahren AT %IX817.0 : BOOL;	(*  ~ {LinkedWith:TIID^Gerät 1 (EtherCAT)^A160 (EP2338-0001)^Channel 2^.zyl_rafo_kamm.fb.e_sensor1_ausgefahren} *)
	.zyl_rafo_kamm.fb.e_sensor2_eingefahren AT %IX817.1 : BOOL;
	.zyl_rafo_kamm.fb.e_sensor2_ausgefahren AT %IX817.2 : BOOL;
	.zyl_rafo_kamm.fb.e_sensor3_eingefahren AT %IX817.3 : BOOL;
	.zyl_rafo_kamm.fb.e_sensor3_ausgefahren AT %IX817.4 : BOOL;
	.zyl_rafo_kamm.fb.e_sensor_mittegefahren AT %IX817.5 : BOOL;
	.zyl_rafo_kamm.fb.e_taste_einfahren AT %IX817.6 : BOOL;
	.zyl_rafo_kamm.fb.e_taste_ausfahren AT %IX817.7 : BOOL;
	.zyl_rafo_kamm.fb.a_ventil_einfahren AT %QX750.7 : BOOL;	(*  ~ {LinkedWith:TIID^Gerät 1 (EtherCAT)^A150 (EP2338-0001)^Channel 1^.zyl_rafo_kamm.fb.a_ventil_einfahren} *)
	.zyl_rafo_kamm.fb.a_ventil_ausfahren AT %QX751.0 : BOOL;	(*  ~ {LinkedWith:TIID^Gerät 1 (EtherCAT)^A150 (EP2338-0001)^Channel 2^.zyl_rafo_kamm.fb.a_ventil_ausfahren} *)
